	{attribute 'TcIecLibraryType'}
	{attribute 'external_name' := 'F_VN_MeasureAngleBetweenEdgesExp_GUID_AE732A2F_0C2A_0A0F_674F_B2AA43375E72'}
	(* Measure the angle between 2 edges. *)
	FUNCTION F_VN_MeasureAngleBetweenEdgesExp : HRESULT
	VAR_INPUT
		ipSrcImage	:	ITcVnImage;	(* Source image (1 channel) *)
		fAngle	:	REFERENCE TO REAL;	(* Returns the angle between the detected edges (radians or degrees, depending on bAngleInDegrees) *)
		aInnerPoint	:	REFERENCE TO TcVnPoint2_REAL;	(* Position inside the angle to measure, from which to start the edge search process (in the direction of aOuterPoint1 and aOuterPoint2) *)
		aOuterPoint1	:	REFERENCE TO TcVnPoint2_REAL;	(* Position where the search process for edge 1 ends *)
		aOuterPoint2	:	REFERENCE TO TcVnPoint2_REAL;	(* Position where the search process for edge 2 ends *)
		eEdgeDirection	:	ETcVnEdgeDirection;	(* Specification of the edge direction from aInnerPoint to aOuterPoint1 and aOuterPoint2 to search for *)
		fMinStrength	:	REAL;	(* Specification of the minimum strength (intensity difference) of the edge to search for *)
		nSearchLines	:	UDINT;	(* Width of the search window, i.e. the number of search lines (3, 5, 7, ...), centered around the line specified by aInnerPoint and aOuterPoint1, aOuterPoint2 *)
		fSearchLineDist	:	REAL;	(* Distance between the search lines in pixels (> 0) *)
		nMaxThickness	:	UDINT;	(* Specification of the maximum thickness of the edge to search for, which means fMinStrength must be reached within nMaxThickness pixels *)
		bInvertSearchDirection	:	BOOL;	(* If true, the search starts from each aOuterPoint in direction of aInnerPoint *)
		nSubpixelsIterations	:	UDINT;	(* Specifies the number of subpixels (for INTERPOLATION, 10 - 20 usually is sufficient) or maximum number of iterations for optimizing the parameters (for APPROX_ERF and APPROX_GAUSSIAN, 50 - 100 usually is sufficient) *)
		bAngleInDegrees	:	BOOL;	(* fAngle is in degrees, if true *)
		fApproxPrecision	:	REAL;	(* Specifies the approximation precision for APPROX_ERF and APPROX_GAUSSIAN (0.001 usually is sufficient, unused for INTERPOLATION) *)
		eAlgorithm	:	ETcVnEdgeDetectionAlgorithm;	(* Selection of the edge detection algorithm *)
		ipEdgePoints1	:	REFERENCE TO ITcVnContainer;	(* Returns the detected edge points between aInnerPoint and aOuterPoint1 (ContainerType_Vector_TcVnPoint2_REAL) *)
		ipEdgePoints2	:	REFERENCE TO ITcVnContainer;	(* Returns the detected edge points between aInnerPoint and aOuterPoint2 (ContainerType_Vector_TcVnPoint2_REAL) *)
		hrPrev	:	HRESULT;	(* HRESULT indicating the result of previous operations (If SUCCEEDED(hrPrev) equals false, no operation is executed.) *)
	END_VAR

END_FUNCTION

// Functions/Measurement/F_VN_MeasureEdgeDistance

	{attribute 'TcIecLibraryType'}
	{attribute 'external_name' := 'F_VN_MeasureEdgeDistance_GUID_7CBEE0F0_467B_0047_5A97_FA055498E2F6'}
	(* Measure the distance between 2 parallel edges, using an interpolation method. *)
	FUNCTION F_VN_MeasureEdgeDistance : HRESULT
	VAR_INPUT
		ipSrcImage	:	ITcVnImage;	(* Source image (1 channel) *)
		fAvgDistance	:	REFERENCE TO REAL;	(* Returns the average distance between the detected edges *)
		aStartPoint	:	REFERENCE TO TcVnPoint2_REAL;	(* Position from which to start the search process (in the direction of aEndPoint) *)
		aEndPoint	:	REFERENCE TO TcVnPoint2_REAL;	(* Position where the search process ends *)
		eEdgeDirection	:	ETcVnEdgeDirection;	(* Specification of the edge direction from aStartPoint to aEndPoint to search for *)
		fMinStrength	:	REAL;	(* Specification of the minimum strength (intensity difference) of the edge to search for *)
		nSearchLines	:	UDINT;	(* Width of the search window, i.e. the number of search lines (1, 3, 5, 7, ...), centered around the line specified by aStartPoint and aEndPoint *)
		hrPrev	:	HRESULT;	(* HRESULT indicating the result of previous operations (If SUCCEEDED(hrPrev) equals false, no operation is executed.) *)
	END_VAR

END_FUNCTION

// Functions/Measurement/F_VN_MeasureEdgeDistanceExp

	{attribute 'TcIecLibraryType'}
	{attribute 'external_name' := 'F_VN_MeasureEdgeDistanceExp_GUID_A22933CA_C8EC_0EED_56A6_BA58A31C374F'}
	(* Measure the distance between 2 parallel edges. (expert function) *)
	FUNCTION F_VN_MeasureEdgeDistanceExp : HRESULT
	VAR_INPUT
		ipSrcImage	:	ITcVnImage;	(* Source image (1 channel) *)
		fAvgDistance	:	REFERENCE TO REAL;	(* Returns the average distance between the detected edges *)
		aStartPoint	:	REFERENCE TO TcVnPoint2_REAL;	(* Position from which to start the search process (in the direction of aEndPoint) *)
		aEndPoint	:	REFERENCE TO TcVnPoint2_REAL;	(* Position where the search process ends *)
		eEdgeDirection	:	ETcVnEdgeDirection;	(* Specification of the edge direction from aStartPoint to aEndPoint to search for *)
		fMinStrength	:	REAL;	(* Specification of the minimum strength (intensity difference) of the edge to search for *)
		nSearchLines	:	UDINT;	(* Width of the search window, i.e. the number of search lines (1, 3, 5, 7, ...), centered around the line specified by aStartPoint and aEndPoint *)
		fSearchLineDist	:	REAL;	(* Distance between the search lines in pixels (> 0) *)
		nMaxThickness	:	UDINT;	(* Specification of the maximum thickness of the edge to search for, which means fMinStrength must be reached within nMaxThickness pixels *)
		bInvertSearchDirection	:	BOOL;	(* If true, the search starts from the center point between aStartPoint and aEndPoint in both directions *)
		fSearchGap	:	REAL;	(* Optional width of a gap (>= 0, centered between aStartPoint and aEndPoint), that is neglected for searching edges (can reduce execution time). The 2 edges to search for must be on different sides of the gap. *)
		nSubpixelsIterations	:	UDINT;	(* Specifies the number of subpixels (for INTERPOLATION, 10 - 20 usually is sufficient) or maximum number of iterations for optimizing the parameters (for APPROX_ERF and APPROX_GAUSSIAN, 50 - 100 usually is sufficient) *)
		fApproxPrecision	:	REAL;	(* Specifies the approximation precision for APPROX_ERF and APPROX_GAUSSIAN (0.001 usually is sufficient, unused for INTERPOLATION) *)
		eAlgorithm	:	ETcVnEdgeDetectionAlgorithm;	(* Selection of the edge detection algorithm *)
		ipEdgePoints1	:	REFERENCE TO ITcVnContainer;	(* Returns the detected edge points of the edge near aStartPoint (optional, set to 0 if not required; ContainerType_Vector_TcVnPoint2_REAL) *)
		ipEdgePoints2	:	REFERENCE TO ITcVnContainer;	(* Returns the detected edge points of the edge near aEndPoint (optional, set to 0 if not required; ContainerType_Vector_TcVnPoint2_REAL) *)
		ipDistances	:	REFERENCE TO ITcVnContainer;	(* Returns the distances between the detected edge points (optional, set to 0 if not required; ContainerType_Vector_REAL) *)
		hrPrev	:	HRESULT;	(* HRESULT indicating the result of previous operations (If SUCCEEDED(hrPrev) equals false, no operation is executed.) *)
	END_VAR

END_FUNCTION

// Functions/Measurement/F_VN_MeasureMinEdgeDistance

	{attribute 'TcIecLibraryType'}
	{attribute 'external_name' := 'F_VN_MeasureMinEdgeDistance_GUID_BAEABED5_95CB_0A35_52C1_670B9836C077'}
	(* Measure the minimum distance within the specified search window between 2 edges, using an interpolation method. *)
	FUNCTION F_VN_MeasureMinEdgeDistance : HRESULT
	VAR_INPUT
		ipSrcImage	:	ITcVnImage;	(* Source image (1 channel) *)
		fMinDistance	:	REFERENCE TO REAL;	(* Returns the minimum distance between the detected edges *)
		aStartPoint	:	REFERENCE TO TcVnPoint2_REAL;	(* Position from which to start the search process (in the direction of aEndPoint) *)
		aEndPoint	:	REFERENCE TO TcVnPoint2_REAL;	(* Position where the search process ends *)
		eEdgeDirection	:	ETcVnEdgeDirection;	(* Specification of the edge direction from aStartPoint to aEndPoint to search for *)
		fMinStrength	:	REAL;	(* Specification of the minimum strength (intensity difference) of the edge to search for *)
		nSearchLines	:	UDINT;	(* Width of the search window, i.e. the number of search lines (1, 3, 5, 7, ...), centered around the line specified by aStartPoint and aEndPoint *)
		hrPrev	:	HRESULT;	(* HRESULT indicating the result of previous operations (If SUCCEEDED(hrPrev) equals false, no operation is executed.) *)
	END_VAR

END_FUNCTION

// Functions/Measurement/F_VN_MeasureMinEdgeDistanceExp

	{attribute 'TcIecLibraryType'}
	{attribute 'external_name' := 'F_VN_MeasureMinEdgeDistanceExp_GUID_0C472EFC_B706_0DF3_5CDC_D468A697A380'}
	(* Measure the minimum distance within the specified search window between 2 edges. (expert function) *)
	FUNCTION F_VN_MeasureMinEdgeDistanceExp : HRESULT
	VAR_INPUT
		ipSrcImage	:	ITcVnImage;	(* Source image (1 channel) *)
		fMinDistance	:	REFERENCE TO REAL;	(* Returns the minimum distance between the detected edges *)
		aStartPoint	:	REFERENCE TO TcVnPoint2_REAL;	(* Position from which to start the search process (in the direction of aEndPoint) *)
		aEndPoint	:	REFERENCE TO TcVnPoint2_REAL;	(* Position where the search process ends *)
		eEdgeDirection	:	ETcVnEdgeDirection;	(* Specification of the edge direction from aStartPoint to aEndPoint to search for *)
		fMinStrength	:	REAL;	(* Specification of the minimum strength (intensity difference) of the edge to search for *)
		nSearchLines	:	UDINT;	(* Width of the search window, i.e. the number of search lines (1, 3, 5, 7, ...), centered around the line specified by aStartPoint and aEndPoint *)
		fSearchLineDist	:	REAL;	(* Distance between the search lines in pixels (> 0) *)
		nMaxThickness	:	UDINT;	(* Specification of the maximum thickness of the edge to search for, which means fMinStrength must be reached within nMaxThickness pixels *)
		bInvertSearchDirection	:	BOOL;	(* If true, the search starts from the center point between aStartPoint and aEndPoint in both directions *)
		fSearchGap	:	REAL;	(* Optional width of a gap (>= 0, centered between aStartPoint and aEndPoint), that is neglected for searching edges (can reduce execution time). The 2 edges to search for must be on different sides of the gap. *)
		nSubpixelsIterations	:	UDINT;	(* Specifies the number of subpixels (for INTERPOLATION, 10 - 20 usually is sufficient) or maximum number of iterations for optimizing the parameters (for APPROX_ERF and APPROX_GAUSSIAN, 50 - 100 usually is sufficient) *)
		fApproxPrecision	:	REAL;	(* Specifies the approximation precision for APPROX_ERF and APPROX_GAUSSIAN (0.001 usually is sufficient, unused for INTERPOLATION) *)
		eAlgorithm	:	ETcVnEdgeDetectionAlgorithm;	(* Selection of the edge detection algorithm *)
		ipEdgePoints1	:	REFERENCE TO ITcVnContainer;	(* Returns the detected edge points of the edge near aStartPoint (optional, set to 0 if not required; ContainerType_Vector_TcVnPoint2_REAL) *)
		ipEdgePoints2	:	REFERENCE TO ITcVnContainer;	(* Returns the detected edge points of the edge near aEndPoint (optional, set to 0 if not required; ContainerType_Vector_TcVnPoint2_REAL) *)
		aPoint1	:	REFERENCE TO TcVnPoint2_REAL;	(* Returns the point on the edge near aStartPoint, for which the minimum distance is achieved *)
		aPoint2	:	REFERENCE TO TcVnPoint2_REAL;	(* Returns the point on the edge near aEndPoint, for which the minimum distance is achieved *)
		hrPrev	:	HRESULT;	(* HRESULT indicating the result of previous operations (If SUCCEEDED(hrPrev) equals false, no operation is executed.) *)
	END_VAR

END_FUNCTION

// Functions/Basic Container Operations/F_VN_AdvanceIterator

	{attribute 'TcIecLibraryType'}
	{attribute 'external_name' := 'F_VN_AdvanceIterator_GUID_ACC8E97D_98FD_0CAF_65B6_42FD1B5BC612'}
	(* Advance an iterator by the specified offset. *)
	FUNCTION F_VN_AdvanceIterator : HRESULT
	VAR_INPUT
		ipIterator	:	ITcVnForwardIterator;	(* Iterator to be advanced *)
		nOffset	:	LINT;	(* Offset, by which ipIterator is advanced *)
		hrPrev	:	HRESULT;	(* HRESULT indicating the result of previous operations (If SUCCEEDED(hrPrev) equals false, no operation is executed.) *)
	END_VAR

END_FUNCTION

// Functions/Basic Container Operations/F_VN_CheckIfEmpty

	{attribute 'TcIecLibraryType'}
	{attribute 'external_name' := 'F_VN_CheckIfEmpty_GUID_F72A904D_F5AF_0726_5092_69B65BB6D2D0'}
	(* Checks if the container is empty. (Alternatively use interface method .CheckIfEmpty.) *)
	FUNCTION F_VN_CheckIfEmpty : HRESULT
	VAR_INPUT
		ipContainer	:	ITcVnContainer;	(* Container *)
		hrPrev	:	HRESULT;	(* HRESULT indicating the result of previous operations (If SUCCEEDED(hrPrev) equals false, no operation is executed.) *)
	END_VAR

END_FUNCTION

// Functions/Basic Container Operations/F_VN_CheckIfIteratorIsAtEnd

	{attribute 'TcIecLibraryType'}
	{attribute 'external_name' := 'F_VN_CheckIfIteratorIsAtEnd_GUID_30C2C0F0_70D6_0795_4B1A_E8C5B6524E93'}
	(* Checks if the iterator points to the past-the-end element. (Alternatively use interface method .CheckIfEnd.) *)
	FUNCTION F_VN_CheckIfIteratorIsAtEnd : HRESULT
	VAR_INPUT
		ipIterator	:	ITcVnForwardIterator;	(* Iterator *)
		hrPrev	:	HRESULT;	(* HRESULT indicating the result of previous operations (If SUCCEEDED(hrPrev) equals false, no operation is executed.) *)
	END_VAR

END_FUNCTION

// Functions/Basic Container Operations/F_VN_ConvertContainerType

	{attribute 'TcIecLibraryType'}
	{attribute 'external_name' := 'F_VN_ConvertContainerType_GUID_01A1FD6A_9814_007F_619D_D5C12B443F08'}
	(* Converts a container to another type (Struct element types are not supported). *)
	FUNCTION F_VN_ConvertContainerType : HRESULT
	VAR_INPUT
		ipSrcContainer	:	ITcVnContainer;	(* Source container *)
		ipDestContainer	:	REFERENCE TO ITcVnContainer;	(* Returns the converted container *)
		nDestTypeGuid	:	GUID;	(* Specifies the destination container type for the conversion *)
		hrPrev	:	HRESULT;	(* HRESULT indicating the result of previous operations (If SUCCEEDED(hrPrev) equals false, no operation is executed.) *)
	END_VAR

END_FUNCTION

// Functions/Basic Container Operations/F_VN_CopyContainer

	{attribute 'TcIecLibraryType'}
	{attribute 'external_name' := 'F_VN_CopyContainer_GUID_DAA3A3C5_5EBA_03BD_7F09_6558B2F826E3'}
	(* Copys a container. *)
	FUNCTION F_VN_CopyContainer : HRESULT
	VAR_INPUT
		ipSrcContainer	:	ITcVnContainer;	(* Source container *)
		ipDestContainer	:	REFERENCE TO ITcVnContainer;	(* Destination container (same type ID as ipSrcContainer; Non-zero interface pointers are reused.) *)
		hrPrev	:	HRESULT;	(* HRESULT indicating the result of previous operations (If SUCCEEDED(hrPrev) equals false, no operation is executed.) *)
	END_VAR

END_FUNCTION

// Functions/Basic Container Operations/F_VN_CopyContainerElementsConditional_ITcVnContainer

	{attribute 'TcIecLibraryType'}
	{attribute 'external_name' := 'F_VN_CopyContainerElementsConditional_ITcVnContainer_GUID_2F464D18_7218_035A_4EBD_E5C0F488799D'}
	(* Copys container elements to a new container, depending on a custom condition. *)
	FUNCTION F_VN_CopyContainerElementsConditional_ITcVnContainer : HRESULT
	VAR_INPUT
		ipSrcContainer	:	ITcVnContainer;	(* Source container *)
		ipDestContainer	:	REFERENCE TO ITcVnContainer;	(* Returns a container with elements, that match the condition *)
		ipConditionFB	:	ITcVnCustomElementCondition_ITcVnContainer;	(* Custom condition *)
		hrPrev	:	HRESULT;	(* HRESULT indicating the result of previous operations (If SUCCEEDED(hrPrev) equals false, no operation is executed.) *)
	END_VAR

END_FUNCTION

// Interfaces/Containers/Function Blocks/ITcVnCustomElementCondition_ITcVnContainer

	(* Offers an interface for a custom condition computed for a container. *)
	{attribute 'c++_compatible'}
	INTERFACE ITcVnCustomElementCondition_ITcVnContainer


(* Evaluates the condition for the container. *)
	{attribute 'c++_compatible'}
	{attribute 'minimal_input_size' := '4'}
	{attribute 'pack_mode' := '4'}
	METHOD Condition : BOOL
	VAR_INPUT
		ipElement : ITcVnContainer;
	END_VAR
END_METHOD

END_INTERFACE

// Functions/Basic Container Operations/F_VN_CopyContainerElementsConditional_ITcVnForwardIterator

	{attribute 'TcIecLibraryType'}
	{attribute 'external_name' := 'F_VN_CopyContainerElementsConditional_ITcVnForwardIterator_GUID_435C1609_A638_0537_49B4_06CAF8EA0EB5'}
	(* Copys container elements to a new container, depending on a custom condition. *)
	FUNCTION F_VN_CopyContainerElementsConditional_ITcVnForwardIterator : HRESULT
	VAR_INPUT
		ipSrcContainer	:	ITcVnContainer;	(* Source container *)
		ipDestContainer	:	REFERENCE TO ITcVnContainer;	(* Returns a container with elements, that match the condition *)
		ipConditionFB	:	ITcVnCustomElementCondition_ITcVnForwardIterator;	(* Custom condition *)
		hrPrev	:	HRESULT;	(* HRESULT indicating the result of previous operations (If SUCCEEDED(hrPrev) equals false, no operation is executed.) *)
	END_VAR

END_FUNCTION

// Interfaces/Containers/Function Blocks/ITcVnCustomElementCondition_ITcVnForwardIterator

	(* Offers an interface for a custom condition computed for an element represented by an ITcVnForwardIterator. *)
	{attribute 'c++_compatible'}
	INTERFACE ITcVnCustomElementCondition_ITcVnForwardIterator


(* Evaluates the condition for the provided element. *)
	{attribute 'c++_compatible'}
	{attribute 'minimal_input_size' := '4'}
	{attribute 'pack_mode' := '4'}
	METHOD Condition : BOOL
	VAR_INPUT
		ipElement : ITcVnForwardIterator;
	END_VAR
END_METHOD

END_INTERFACE

// Functions/Basic Container Operations/F_VN_CreateContainer

	{attribute 'TcIecLibraryType'}
	{attribute 'external_name' := 'F_VN_CreateContainer_GUID_61D37913_CA0D_07D0_5304_6E5DDCD021C0'}
	(* Creates a container with type GUID nTypeGuid and return its container interface. *)
	FUNCTION F_VN_CreateContainer : HRESULT
	VAR_INPUT
		ipContainer	:	REFERENCE TO ITcVnContainer;	(* Returns the created container *)
		nTypeGuid	:	GUID;	(* Type GUID of the container to be created *)
		nElementNum	:	ULINT;	(* Number of elements *)
		hrPrev	:	HRESULT;	(* HRESULT indicating the result of previous operations (If SUCCEEDED(hrPrev) equals false, no operation is executed.) *)
	END_VAR

END_FUNCTION

// Functions/Basic Container Operations/F_VN_CreateContainerFromArray

	{attribute 'TcIecLibraryType'}
	{attribute 'external_name' := 'F_VN_CreateContainerFromArray_GUID_AA5B3DDF_00B1_0B21_7AD4_970908632B01'}
	(* Creates a container with type GUID nTypeGuid, initialize it with provided data and return its container interface. Only supported for basic container types, i.e. not for containers of containers. *)
	FUNCTION F_VN_CreateContainerFromArray : HRESULT
	VAR_INPUT
		pData	:	PVOID;	(* Pointer to the data array. Make sure that the array contains at least nElementNum elements and that the array element type matches the container element type. *)
		ipContainer	:	REFERENCE TO ITcVnContainer;	(* Returns the created container *)
		nTypeGuid	:	GUID;	(* Type GUID of the container to be created *)
		nElementNum	:	ULINT;	(* Number of elements to copy from pData *)
		hrPrev	:	HRESULT;	(* HRESULT indicating the result of previous operations (If SUCCEEDED(hrPrev) equals false, no operation is executed.) *)
	END_VAR

END_FUNCTION

// Functions/Basic Container Operations/F_VN_EraseFromContainer

	{attribute 'TcIecLibraryType'}
	{attribute 'external_name' := 'F_VN_EraseFromContainer_GUID_D686421B_0E77_0897_58AA_85FC33B178E9'}
	(* Erase elements from a container. *)
	FUNCTION F_VN_EraseFromContainer : HRESULT
	VAR_INPUT
		ipContainer	:	ITcVnContainer;	(* Container from which to erase elements *)
		nStartIdx	:	ULINT;	(* Index of the first element to erase *)
		nCount	:	ULINT;	(* Number of elements to erase *)
		hrPrev	:	HRESULT;	(* HRESULT indicating the result of previous operations (If SUCCEEDED(hrPrev) equals false, no operation is executed.) *)
	END_VAR

END_FUNCTION

// Functions/Basic Container Operations/F_VN_ExportContainer

	{attribute 'TcIecLibraryType'}
	{attribute 'external_name' := 'F_VN_ExportContainer_GUID_B3105DE8_989A_095E_6EB1_2DCFC3551E31'}
	(* Export the container elements into a buffer (e.g. an array). Only possible for containers with basic elements. *)
	FUNCTION F_VN_ExportContainer : HRESULT
	VAR_INPUT
		ipContainer	:	ITcVnContainer;	(* Container with basic elements *)
		pBuffer	:	PVOID;	(* Buffer to store the container elements (Make sure to allocate enough memory! The required size in bytes can be determined using the function F_VN_ExportContainerSize) *)
		nBufferSize	:	ULINT;	(* Size of the buffer memory in bytes *)
		hrPrev	:	HRESULT;	(* HRESULT indicating the result of previous operations (If SUCCEEDED(hrPrev) equals false, no operation is executed.) *)
	END_VAR

END_FUNCTION

// Functions/Basic Container Operations/F_VN_ExportContainerSize

	{attribute 'TcIecLibraryType'}
	{attribute 'external_name' := 'F_VN_ExportContainerSize_GUID_76F4BBB5_BAC4_061D_63B1_EE647B621371'}
	(* Determine the required buffer size in bytes to store all container elements (number_of_Elements * size_per_Element). Only possible for containers with basic elements. *)
	FUNCTION F_VN_ExportContainerSize : HRESULT
	VAR_INPUT
		ipContainer	:	ITcVnContainer;	(* Container with basic elements *)
		nBufferSize	:	REFERENCE TO ULINT;	(* Output parameter containing the required buffer size *)
		hrPrev	:	HRESULT;	(* HRESULT indicating the result of previous operations (If SUCCEEDED(hrPrev) equals false, no operation is executed.) *)
	END_VAR

END_FUNCTION

// Functions/Basic Container Operations/F_VN_ExportContainer_String

	{attribute 'TcIecLibraryType'}
	{attribute 'external_name' := 'F_VN_ExportContainer_String_GUID_5BD8ABC1_1BA1_0734_5AF1_0620F612769A'}
	(* Export the container elements into a string. Only possible for containers of type ContainerType_String_SINT. *)
	FUNCTION F_VN_ExportContainer_String : HRESULT
	VAR_INPUT
		ipContainer	:	ITcVnContainer;	(* Container of type ContainerType_String_SINT *)
	END_VAR
	VAR_IN_OUT CONSTANT
		sText	:	STRING;	(* Make sure to choose a sufficient STRING size! The required size can be determined using the function VnExportContainerSize. *)
	END_VAR
	VAR_INPUT
		nMaxLength	:	ULINT;	(* Maximum string length to export (including 0 termination). If the container content is longer, the string is cut off at nMaxLength - 1 and 0 termination is appended. In this case, S_FALSE is returned. *)
		hrPrev	:	HRESULT;	(* HRESULT indicating the result of previous operations (If SUCCEEDED(hrPrev) equals false, no operation is executed.) *)
	END_VAR

END_FUNCTION

// Functions/Basic Container Operations/F_VN_ExportSubContainer

	{attribute 'TcIecLibraryType'}
	{attribute 'external_name' := 'F_VN_ExportSubContainer_GUID_2C76D183_CD1A_0BBB_4C3C_54CD9386FE08'}
	(* Export the container elements of a sub-container into a buffer (e.g. an array). Only possible for 2-dimensional containers with basic elements. *)
	FUNCTION F_VN_ExportSubContainer : HRESULT
	VAR_INPUT
		ipContainer	:	ITcVnContainer;	(* Container with basic elements *)
		nIndex	:	ULINT;	(* Index of the requested element *)
		pBuffer	:	PVOID;	(* Buffer to store the container elements (Make sure to allocate enough memory! The required size in bytes can be determined using the function F_VN_ExportSubContainerSize) *)
		nBufferSize	:	ULINT;	(* Size of the buffer memory in bytes *)
		hrPrev	:	HRESULT;	(* HRESULT indicating the result of previous operations (If SUCCEEDED(hrPrev) equals false, no operation is executed.) *)
	END_VAR

END_FUNCTION

// Functions/Basic Container Operations/F_VN_ExportSubContainerSize

	{attribute 'TcIecLibraryType'}
	{attribute 'external_name' := 'F_VN_ExportSubContainerSize_GUID_9A378173_3E8F_041B_7D7A_DBB1303321B8'}
	(* Determine the required buffer size in bytes to store all container elements of a sub-container (number_of_Elements * size_per_Element). Only possible for 2-dimensional containers with basic elements. *)
	FUNCTION F_VN_ExportSubContainerSize : HRESULT
	VAR_INPUT
		ipContainer	:	ITcVnContainer;	(* Container with basic elements *)
		nIndex	:	ULINT;	(* Index of the requested element *)
		nBufferSize	:	REFERENCE TO ULINT;	(* Output parameter containing the required buffer size *)
		hrPrev	:	HRESULT;	(* HRESULT indicating the result of previous operations (If SUCCEEDED(hrPrev) equals false, no operation is executed.) *)
	END_VAR

END_FUNCTION

// Functions/Basic Container Operations/F_VN_ExportSubContainer_String

	{attribute 'TcIecLibraryType'}
	{attribute 'external_name' := 'F_VN_ExportSubContainer_String_GUID_4F555A08_F7D7_0928_7E2C_5AC3BF1C3727'}
	(* Export the container elements of a sub-container into a string. Only possible for 2-dimensional containers of type ContainerType_Vector_String_SINT. *)
	FUNCTION F_VN_ExportSubContainer_String : HRESULT
	VAR_INPUT
		ipContainer	:	ITcVnContainer;	(* Container of type ContainerType_Vector_String_SINT *)
		nIndex	:	ULINT;	(* Index of the requested element *)
	END_VAR
	VAR_IN_OUT CONSTANT
		sText	:	STRING;	(* Make sure to choose a sufficient STRING size! The required size can be determined using the function VnExportSubContainerSize. *)
	END_VAR
	VAR_INPUT
		nMaxLength	:	ULINT;	(* Maximum string length to export (including 0 termination). If the container content is longer, the string is cut off at nMaxLength - 1 and 0 termination is appended. In this case, S_FALSE is returned. *)
		hrPrev	:	HRESULT;	(* HRESULT indicating the result of previous operations (If SUCCEEDED(hrPrev) equals false, no operation is executed.) *)
	END_VAR

END_FUNCTION

// Functions/Basic Container Operations/F_VN_ExtractContainerRange

	{attribute 'TcIecLibraryType'}
	{attribute 'external_name' := 'F_VN_ExtractContainerRange_GUID_4EB284E8_0B53_0D83_5DCE_29B545B8D0A0'}
	(* Copy the specified range of the source container into the destination container. (If the destination container already contains elements, they will be removed.) *)
	FUNCTION F_VN_ExtractContainerRange : HRESULT
	VAR_INPUT
		ipSrcContainer	:	ITcVnContainer;	(* Source container *)
		ipDestContainer	:	REFERENCE TO ITcVnContainer;	(* Destination container *)
		nFirstIdx	:	ULINT;	(* Index of the first element to copy *)
		nLastIdx	:	ULINT;	(* Index of the last element to copy *)
		hrPrev	:	HRESULT;	(* HRESULT indicating the result of previous operations (If SUCCEEDED(hrPrev) equals false, no operation is executed.) *)
	END_VAR

END_FUNCTION

// Functions/Basic Container Operations/F_VN_GetContainer

	{attribute 'TcIecLibraryType'}
	{attribute 'external_name' := 'F_VN_GetContainer_GUID_27505B6E_9EAE_086D_5BCA_CC9172BAFD0B'}
	(* Gets a pointer to the current element converted into an ITcVnContainer interface and increment its reference counter (only possible for container types). (Alternatively use interface method .GetContainer.) *)
	FUNCTION F_VN_GetContainer : HRESULT
	VAR_INPUT
		ipIterator	:	ITcVnForwardIterator;	(* Iterator *)
		ipContainer	:	REFERENCE TO ITcVnContainer;	(* Returns the container interface *)
		hrPrev	:	HRESULT;	(* HRESULT indicating the result of previous operations (If SUCCEEDED(hrPrev) equals false, no operation is executed.) *)
	END_VAR

END_FUNCTION

// Functions/Basic Container Operations/F_VN_GetContainerExp

	{attribute 'TcIecLibraryType'}
	{attribute 'external_name' := 'F_VN_GetContainerExp_GUID_436CF1E3_F353_08D3_710A_C75CD81D8DEB'}
	(* Gets a pointer to the current element converted into an ITcVnContainer interface and increment its reference counter (only possible for container types). Additionally, an offset to increment or decrement the iterator afterwards can be provided. (expert function) *)
	FUNCTION F_VN_GetContainerExp : HRESULT
	VAR_INPUT
		ipIterator	:	ITcVnForwardIterator;	(* Iterator *)
		ipContainer	:	REFERENCE TO ITcVnContainer;	(* Returns the container interface *)
		nOffset	:	DINT;	(* Offset to increment (>0) or decrement (<0) the iterator afterwards *)
		hrPrev	:	HRESULT;	(* HRESULT indicating the result of previous operations (If SUCCEEDED(hrPrev) equals false, no operation is executed.) *)
	END_VAR

END_FUNCTION

// Functions/Basic Container Operations/F_VN_GetForwardIterator

	{attribute 'TcIecLibraryType'}
	{attribute 'external_name' := 'F_VN_GetForwardIterator_GUID_43078F70_57B1_0E73_4856_F4D286EF9EA2'}
	(* Gets a forward iterator for the container. (Alternatively use interface method .GetForwardIterator.) *)
	FUNCTION F_VN_GetForwardIterator : HRESULT
	VAR_INPUT
		ipContainer	:	ITcVnContainer;	(* Container *)
		ipIterator	:	REFERENCE TO ITcVnForwardIterator;	(* Returns the iterator interface *)
		hrPrev	:	HRESULT;	(* HRESULT indicating the result of previous operations (If SUCCEEDED(hrPrev) equals false, no operation is executed.) *)
	END_VAR

END_FUNCTION

// Functions/Basic Container Operations/F_VN_GetNumberOfElements

	{attribute 'TcIecLibraryType'}
	{attribute 'external_name' := 'F_VN_GetNumberOfElements_GUID_C1684A08_CB59_09CF_7B51_7659520AA3E9'}
	(* Gets the number of elements in the container. (Alternatively use interface method .getElementNum.) *)
	FUNCTION F_VN_GetNumberOfElements : HRESULT
	VAR_INPUT
		ipContainer	:	ITcVnContainer;	(* Container *)
		nNumberOfElements	:	REFERENCE TO ULINT;	(* Returns the number of elements in ipContainer *)
		hrPrev	:	HRESULT;	(* HRESULT indicating the result of previous operations (If SUCCEEDED(hrPrev) equals false, no operation is executed.) *)
	END_VAR

END_FUNCTION

// Functions/Basic Container Operations/F_VN_GetRandomAccessIterator

	{attribute 'TcIecLibraryType'}
	{attribute 'external_name' := 'F_VN_GetRandomAccessIterator_GUID_3FA92340_67E8_032A_7ED0_6A69355C56A7'}
	(* Gets a random access iterator for the container. (Alternatively use interface method .GetRandomAccessIterator.) *)
	FUNCTION F_VN_GetRandomAccessIterator : HRESULT
	VAR_INPUT
		ipContainer	:	ITcVnContainer;	(* Container *)
		ipIterator	:	REFERENCE TO ITcVnRandomAccessIterator;	(* Returns the iterator interface *)
		hrPrev	:	HRESULT;	(* HRESULT indicating the result of previous operations (If SUCCEEDED(hrPrev) equals false, no operation is executed.) *)
	END_VAR

END_FUNCTION

// Functions/Basic Container Operations/F_VN_IncrementIterator

	{attribute 'TcIecLibraryType'}
	{attribute 'external_name' := 'F_VN_IncrementIterator_GUID_69A16AA6_5F55_058E_6ED7_D592BD9145A4'}
	(* Increment the iterator. (Alternatively use interface method .Increment.) *)
	FUNCTION F_VN_IncrementIterator : HRESULT
	VAR_INPUT
		ipIterator	:	ITcVnForwardIterator;	(* Iterator *)
		hrPrev	:	HRESULT;	(* HRESULT indicating the result of previous operations (If SUCCEEDED(hrPrev) equals false, no operation is executed.) *)
	END_VAR

END_FUNCTION

// Functions/Basic Container Operations/F_VN_IteratorDistance

	{attribute 'TcIecLibraryType'}
	{attribute 'external_name' := 'F_VN_IteratorDistance_GUID_DC10392B_7965_07D5_51DE_916FCBD58C32'}
	(* Computes the distance between 2 iterators. *)
	FUNCTION F_VN_IteratorDistance : HRESULT
	VAR_INPUT
		ipIteratorFirst	:	ITcVnForwardIterator;	(* First iterator *)
		ipIteratorLast	:	ITcVnForwardIterator;	(* Last iterator *)
		nDistance	:	REFERENCE TO LINT;	(* Returns the computed distance *)
		hrPrev	:	HRESULT;	(* HRESULT indicating the result of previous operations (If SUCCEEDED(hrPrev) equals false, no operation is executed.) *)
	END_VAR

END_FUNCTION

// Functions/Basic Container Operations/F_VN_ReserveContainerMemory

	{attribute 'TcIecLibraryType'}
	{attribute 'external_name' := 'F_VN_ReserveContainerMemory_GUID_A6C96216_5A91_0611_6333_23BBD3722D9C'}
	(* Reserve container memory (call with maximum required number of elements before manually appending elements for better performance) *)
	FUNCTION F_VN_ReserveContainerMemory : HRESULT
	VAR_INPUT
		ipContainer	:	ITcVnContainer;	(* Container for which to reserve the memory *)
		nElements	:	ULINT;	(* Number of elements for which the container should reserve memory *)
		hrPrev	:	HRESULT;	(* HRESULT indicating the result of previous operations (If SUCCEEDED(hrPrev) equals false, no operation is executed.) *)
	END_VAR

END_FUNCTION

// Functions/Basic Container Operations/F_VN_ReverseContainer

	{attribute 'TcIecLibraryType'}
	{attribute 'external_name' := 'F_VN_ReverseContainer_GUID_35F112E5_387D_0B85_557A_AEA6C3B2DB12'}
	(* Reverse the container elements. *)
	FUNCTION F_VN_ReverseContainer : HRESULT
	VAR_INPUT
		ipContainer	:	ITcVnContainer;	(* Container to be reversed *)
		hrPrev	:	HRESULT;	(* HRESULT indicating the result of previous operations (If SUCCEEDED(hrPrev) equals false, no operation is executed.) *)
	END_VAR

END_FUNCTION

// Functions/Basic Container Operations/F_VN_SetContainer

	{attribute 'TcIecLibraryType'}
	{attribute 'external_name' := 'F_VN_SetContainer_GUID_E3937A25_D58C_09AB_7741_9A0CBC6B0412'}
	(* Sets the current element using an ITcVnContainer interface (only possible for container types). (Alternatively use interface method .SetContainer.) *)
	FUNCTION F_VN_SetContainer : HRESULT
	VAR_INPUT
		ipIterator	:	ITcVnForwardIterator;	(* Iterator *)
		ipContainer	:	ITcVnContainer;	(* Container interface of which the content is to be assigned to the current element *)
		hrPrev	:	HRESULT;	(* HRESULT indicating the result of previous operations (If SUCCEEDED(hrPrev) equals false, no operation is executed.) *)
	END_VAR

END_FUNCTION

// Functions/Basic Container Operations/F_VN_SetIteratorToBegin

	{attribute 'TcIecLibraryType'}
	{attribute 'external_name' := 'F_VN_SetIteratorToBegin_GUID_51E4D889_EE17_05C3_44C3_7A5207251AFA'}
	(* Sets the iterator to the first element of the container. (Alternatively use interface method .SetToBegin.) *)
	FUNCTION F_VN_SetIteratorToBegin : HRESULT
	VAR_INPUT
		ipIterator	:	ITcVnForwardIterator;	(* Iterator *)
		hrPrev	:	HRESULT;	(* HRESULT indicating the result of previous operations (If SUCCEEDED(hrPrev) equals false, no operation is executed.) *)
	END_VAR

END_FUNCTION

// Functions/Geometric and Coordinate Transformations/F_VN_AlignRotatedImageRegion

	{attribute 'TcIecLibraryType'}
	{attribute 'external_name' := 'F_VN_AlignRotatedImageRegion_GUID_3F265FEA_BECE_014F_47AF_B5F8C6E76B10'}
	(* Copies the provided image region and aligns it to the image axes. *)
	FUNCTION F_VN_AlignRotatedImageRegion : HRESULT
	VAR_INPUT
		ipSrcImage	:	ITcVnImage;	(* Source image *)
		ipDestImage	:	REFERENCE TO ITcVnImage;	(* Destination image (An appropriate image will be created if required.) *)
		stRegion	:	REFERENCE TO TcVnRotatedRectangle;	(* Image region to be aligned *)
		hrPrev	:	HRESULT;	(* HRESULT indicating the result of previous operations (If SUCCEEDED(hrPrev) equals false, no operation is executed.) *)
	END_VAR

END_FUNCTION

// Functions/Geometric and Coordinate Transformations/F_VN_AlignRotatedImageRegionExp

	{attribute 'TcIecLibraryType'}
	{attribute 'external_name' := 'F_VN_AlignRotatedImageRegionExp_GUID_D33A5843_210C_0064_6EBC_CB88CD706C00'}
	(* Copies the provided image region and aligns it to the image axes. (expert function) *)
	FUNCTION F_VN_AlignRotatedImageRegionExp : HRESULT
	VAR_INPUT
		ipSrcImage	:	ITcVnImage;	(* Source image *)
		ipDestImage	:	REFERENCE TO ITcVnImage;	(* Destination image (An appropriate image will be created if required.) *)
		stRegion	:	REFERENCE TO TcVnRotatedRectangle;	(* Image region to be aligned *)
		eInterpolationType	:	ETcVnInterpolationType;	(* Interpolation method *)
		eBorderInterpolation	:	ETcVnBorderInterpolationMethod;	(* Border interpolation method (ISOLATED not supported) *)
		aBorderValue	:	REFERENCE TO TcVnVector4_LREAL;	(* Border value, if CONSTANT is used *)
		hrPrev	:	HRESULT;	(* HRESULT indicating the result of previous operations (If SUCCEEDED(hrPrev) equals false, no operation is executed.) *)
	END_VAR

END_FUNCTION

// Functions/Geometric and Coordinate Transformations/F_VN_ApplyRotationToAffineTransformation

	{attribute 'TcIecLibraryType'}
	{attribute 'external_name' := 'F_VN_ApplyRotationToAffineTransformation_GUID_D2AAEA5C_C5D3_0D46_678A_5DCA00EA5833'}
	(* Apply a rotation to an existing 2D affine transformation matrix. *)
	FUNCTION F_VN_ApplyRotationToAffineTransformation : HRESULT
	VAR_INPUT
		aTransformationMatrix	:	REFERENCE TO TcVnMatrix2x3_LREAL;	(* Affine transformation matrix to which the rotation is applied *)
		fAngle	:	LREAL;	(* Angle in radians (positive means counter-clockwise) *)
		hrPrev	:	HRESULT;	(* HRESULT indicating the result of previous operations (If SUCCEEDED(hrPrev) equals false, no operation is executed.) *)
	END_VAR

END_FUNCTION

// Functions/Geometric and Coordinate Transformations/F_VN_ApplyRotationToAffineTransformationExp

	{attribute 'TcIecLibraryType'}
	{attribute 'external_name' := 'F_VN_ApplyRotationToAffineTransformationExp_GUID_09811113_83D1_0FA5_740A_AEC9964AC26B'}
	(* Apply a rotation to an existing 2D affine transformation matrix. (expert function) *)
	FUNCTION F_VN_ApplyRotationToAffineTransformationExp : HRESULT
	VAR_INPUT
		aTransformationMatrix	:	REFERENCE TO TcVnMatrix2x3_LREAL;	(* Affine transformation matrix to which the rotation is applied *)
		fAngle	:	LREAL;	(* Angle in radians (positive means counter-clockwise) *)
		bUsePreMultiplication	:	BOOL;	(* Select if pre- or post-multiplication should be used *)
		hrPrev	:	HRESULT;	(* HRESULT indicating the result of previous operations (If SUCCEEDED(hrPrev) equals false, no operation is executed.) *)
	END_VAR

END_FUNCTION

// Functions/Geometric and Coordinate Transformations/F_VN_ApplyScalingToAffineTransformation

	{attribute 'TcIecLibraryType'}
	{attribute 'external_name' := 'F_VN_ApplyScalingToAffineTransformation_GUID_0AC37701_099D_0829_772F_D6736195BB34'}
	(* Apply a scaling to an existing 2D affine transformation matrix. *)
	FUNCTION F_VN_ApplyScalingToAffineTransformation : HRESULT
	VAR_INPUT
		aTransformationMatrix	:	REFERENCE TO TcVnMatrix2x3_LREAL;	(* Affine transformation matrix to which the scaling is applied *)
		fScaleX	:	LREAL;	(* Scaling factor in x direction *)
		fScaleY	:	LREAL;	(* Scaling factor in y direction *)
		hrPrev	:	HRESULT;	(* HRESULT indicating the result of previous operations (If SUCCEEDED(hrPrev) equals false, no operation is executed.) *)
	END_VAR

END_FUNCTION

// Functions/Geometric and Coordinate Transformations/F_VN_ApplyScalingToAffineTransformationExp

	{attribute 'TcIecLibraryType'}
	{attribute 'external_name' := 'F_VN_ApplyScalingToAffineTransformationExp_GUID_0B1DCD8E_602D_0379_4AFD_8BE184FF709D'}
	(* Apply a scaling to an existing 2D affine transformation matrix. (expert function) *)
	FUNCTION F_VN_ApplyScalingToAffineTransformationExp : HRESULT
	VAR_INPUT
		aTransformationMatrix	:	REFERENCE TO TcVnMatrix2x3_LREAL;	(* Affine transformation matrix to which the scaling is applied *)
		fScaleX	:	LREAL;	(* Scaling factor in x direction *)
		fScaleY	:	LREAL;	(* Scaling factor in y direction *)
		bUsePreMultiplication	:	BOOL;	(* Select if pre- or post-multiplication should be used *)
		hrPrev	:	HRESULT;	(* HRESULT indicating the result of previous operations (If SUCCEEDED(hrPrev) equals false, no operation is executed.) *)
	END_VAR

END_FUNCTION

// Functions/Geometric and Coordinate Transformations/F_VN_ApplyTranslationToAffineTransformation

	{attribute 'TcIecLibraryType'}
	{attribute 'external_name' := 'F_VN_ApplyTranslationToAffineTransformation_GUID_2CE336D6_8FF6_0659_73D0_7BE4ABCDC41C'}
	(* Apply a translation to an existing 2D affine transformation matrix. *)
	FUNCTION F_VN_ApplyTranslationToAffineTransformation : HRESULT
	VAR_INPUT
		aTransformationMatrix	:	REFERENCE TO TcVnMatrix2x3_LREAL;	(* Affine transformation matrix to which the translation is applied *)
		fDeltaX	:	LREAL;	(* Translation in x direction *)
		fDeltaY	:	LREAL;	(* Translation in y direction *)
		hrPrev	:	HRESULT;	(* HRESULT indicating the result of previous operations (If SUCCEEDED(hrPrev) equals false, no operation is executed.) *)
	END_VAR

END_FUNCTION

// Functions/Geometric and Coordinate Transformations/F_VN_ApplyTranslationToAffineTransformationExp

	{attribute 'TcIecLibraryType'}
	{attribute 'external_name' := 'F_VN_ApplyTranslationToAffineTransformationExp_GUID_B48E036C_FF70_0D75_7B83_23F5D06CED29'}
	(* Apply a translation to an existing 2D affine transformation matrix. (expert function) *)
	FUNCTION F_VN_ApplyTranslationToAffineTransformationExp : HRESULT
	VAR_INPUT
		aTransformationMatrix	:	REFERENCE TO TcVnMatrix2x3_LREAL;	(* Affine transformation matrix to which the translation is applied *)
		fDeltaX	:	LREAL;	(* Translation in x direction *)
		fDeltaY	:	LREAL;	(* Translation in y direction *)
		bUsePreMultiplication	:	BOOL;	(* Select if pre- or post-multiplication should be used *)
		hrPrev	:	HRESULT;	(* HRESULT indicating the result of previous operations (If SUCCEEDED(hrPrev) equals false, no operation is executed.) *)
	END_VAR

END_FUNCTION

// Functions/Geometric and Coordinate Transformations/F_VN_ApplyYAxisInversionToAffineTransformation

	{attribute 'TcIecLibraryType'}
	{attribute 'external_name' := 'F_VN_ApplyYAxisInversionToAffineTransformation_GUID_ABA7B922_0E85_0EC7_45FC_DB03AB370BB3'}
	(* Apply an inversion of the y-axis direction to an existing 2D affine transformation matrix. *)
	FUNCTION F_VN_ApplyYAxisInversionToAffineTransformation : HRESULT
	VAR_INPUT
		aTransformationMatrix	:	REFERENCE TO TcVnMatrix2x3_LREAL;	(* Affine transformation matrix to which the inversion of the y-axis direction is applied *)
		hrPrev	:	HRESULT;	(* HRESULT indicating the result of previous operations (If SUCCEEDED(hrPrev) equals false, no operation is executed.) *)
	END_VAR

END_FUNCTION

// Functions/Geometric and Coordinate Transformations/F_VN_ApplyYAxisInversionToAffineTransformationExp

	{attribute 'TcIecLibraryType'}
	{attribute 'external_name' := 'F_VN_ApplyYAxisInversionToAffineTransformationExp_GUID_0519358C_2F66_032D_63C6_2BC545D0AFB4'}
	(* Apply an inversion of the y-axis direction to an existing 2D affine transformation matrix. (expert function) *)
	FUNCTION F_VN_ApplyYAxisInversionToAffineTransformationExp : HRESULT
	VAR_INPUT
		aTransformationMatrix	:	REFERENCE TO TcVnMatrix2x3_LREAL;	(* Affine transformation matrix to which the inversion of the y-axis direction is applied *)
		bUsePreMultiplication	:	BOOL;	(* Select if pre- or post-multiplication should be used *)
		hrPrev	:	HRESULT;	(* HRESULT indicating the result of previous operations (If SUCCEEDED(hrPrev) equals false, no operation is executed.) *)
	END_VAR

END_FUNCTION

// Functions/Geometric and Coordinate Transformations/F_VN_ConvertCartesianToPolarAngleImage

	{attribute 'TcIecLibraryType'}
	{attribute 'external_name' := 'F_VN_ConvertCartesianToPolarAngleImage_GUID_17EADBBD_F562_070F_5C5C_9C9C6F0DA8B4'}
	(* Converts cartesian coordinates (x, y) to polar angle. *)
	FUNCTION F_VN_ConvertCartesianToPolarAngleImage : HRESULT
	VAR_INPUT
		ipSrcImageX	:	ITcVnImage;	(* Source image containing the x values (elements of type REAL or LREAL) *)
		ipSrcImageY	:	ITcVnImage;	(* Source image containing the y values (Same element type as ipSrcImageX) *)
		ipDestImageAng	:	REFERENCE TO ITcVnImage;	(* Destination image containing the angles (Same element type as source images. An appropriate destination image will be created if required.) *)
		hrPrev	:	HRESULT;	(* HRESULT indicating the result of previous operations (If SUCCEEDED(hrPrev) equals false, no operation is executed.) *)
	END_VAR

END_FUNCTION

// Functions/Geometric and Coordinate Transformations/F_VN_ConvertCartesianToPolarAngleImageExp

	{attribute 'TcIecLibraryType'}
	{attribute 'external_name' := 'F_VN_ConvertCartesianToPolarAngleImageExp_GUID_1D68747B_2AEF_02D8_5804_BAE8BD678C2F'}
	(* Converts cartesian coordinates (x, y) to polar angle. (expert function) *)
	FUNCTION F_VN_ConvertCartesianToPolarAngleImageExp : HRESULT
	VAR_INPUT
		ipSrcImageX	:	ITcVnImage;	(* Source image containing the x values (elements of type REAL or LREAL) *)
		ipSrcImageY	:	ITcVnImage;	(* Source image containing the y values (Same element type as ipSrcImageX) *)
		ipDestImageAng	:	REFERENCE TO ITcVnImage;	(* Destination image containing the angles (Same element type as source images. An appropriate destination image will be created if required.) *)
		bAngleInDegrees	:	BOOL;	(* Specifys, if the angles should be in degrees or radians *)
		hrPrev	:	HRESULT;	(* HRESULT indicating the result of previous operations (If SUCCEEDED(hrPrev) equals false, no operation is executed.) *)
	END_VAR

END_FUNCTION

// Functions/Geometric and Coordinate Transformations/F_VN_ConvertCartesianToPolarAngles

	{attribute 'TcIecLibraryType'}
	{attribute 'external_name' := 'F_VN_ConvertCartesianToPolarAngles_GUID_E7144BB7_132A_0642_64B6_73DCB69099EE'}
	(* Converts cartesian coordinates (x, y) to polar angle. *)
	FUNCTION F_VN_ConvertCartesianToPolarAngles : HRESULT
	VAR_INPUT
		ipSrcPointsCart	:	ITcVnContainer;	(* Container with cartesian points (ContainerType_Vector_TcVnPoint2_DINT or ContainerType_Vector_TcVnPoint2_REAL or ContainerType_Vector_TcVnPoint2_LREAL) *)
		ipDestAngles	:	REFERENCE TO ITcVnContainer;	(* Returns a container which is filled with the angles (ContainerType_Vector_REAL, if source points are of type TcVnPoint2_DINT or TcVnPoint2_REAL; else ContainerType_Vector_LREAL. Non-zero interface pointers are reused.) *)
		hrPrev	:	HRESULT;	(* HRESULT indicating the result of previous operations (If SUCCEEDED(hrPrev) equals false, no operation is executed.) *)
	END_VAR

END_FUNCTION

// Functions/Geometric and Coordinate Transformations/F_VN_ConvertCartesianToPolarAnglesExp

	{attribute 'TcIecLibraryType'}
	{attribute 'external_name' := 'F_VN_ConvertCartesianToPolarAnglesExp_GUID_5114B8BE_DDFA_0141_6749_A3EDE6F2388B'}
	(* Converts cartesian coordinates (x, y) to polar angle. (expert function) *)
	FUNCTION F_VN_ConvertCartesianToPolarAnglesExp : HRESULT
	VAR_INPUT
		ipSrcPointsCart	:	ITcVnContainer;	(* Container with cartesian points (ContainerType_Vector_TcVnPoint2_DINT or ContainerType_Vector_TcVnPoint2_REAL or ContainerType_Vector_TcVnPoint2_LREAL) *)
		ipDestAngles	:	REFERENCE TO ITcVnContainer;	(* Returns a container which is filled with the angles (ContainerType_Vector_REAL, if source points are of type TcVnPoint2_DINT or TcVnPoint2_REAL; else ContainerType_Vector_LREAL. Non-zero interface pointers are reused.) *)
		bAngleInDegrees	:	BOOL;	(* Specify, if the angles should be in degrees or radians *)
		hrPrev	:	HRESULT;	(* HRESULT indicating the result of previous operations (If SUCCEEDED(hrPrev) equals false, no operation is executed.) *)
	END_VAR

END_FUNCTION

// Functions/Geometric and Coordinate Transformations/F_VN_ConvertCartesianToPolarImages

	{attribute 'TcIecLibraryType'}
	{attribute 'external_name' := 'F_VN_ConvertCartesianToPolarImages_GUID_F8BA0872_BC93_0005_5BBA_C12C416537B0'}
	(* Converts cartesian coordinates (x, y) to polar coordinates (magnitude, angle). *)
	FUNCTION F_VN_ConvertCartesianToPolarImages : HRESULT
	VAR_INPUT
		ipSrcImageX	:	ITcVnImage;	(* Source image containing the x values (elements of type REAL or LREAL) *)
		ipSrcImageY	:	ITcVnImage;	(* Source image containing the y values (Same element type as ipSrcImageX) *)
		ipDestImageMag	:	REFERENCE TO ITcVnImage;	(* Destination image containing the magnitudes (Same element type as source images. An appropriate destination image will be created if required.) *)
		ipDestImageAng	:	REFERENCE TO ITcVnImage;	(* Destination image containing the angles (Same element type as source images. An appropriate destination image will be created if required.) *)
		hrPrev	:	HRESULT;	(* HRESULT indicating the result of previous operations (If SUCCEEDED(hrPrev) equals false, no operation is executed.) *)
	END_VAR

END_FUNCTION

// Functions/Geometric and Coordinate Transformations/F_VN_ConvertCartesianToPolarImagesExp

	{attribute 'TcIecLibraryType'}
	{attribute 'external_name' := 'F_VN_ConvertCartesianToPolarImagesExp_GUID_C7CB6E2F_D7A7_01AA_4CF2_0CB9BEF7AE79'}
	(* Converts cartesian coordinates (x, y) to polar coordinates (magnitude, angle). (expert function) *)
	FUNCTION F_VN_ConvertCartesianToPolarImagesExp : HRESULT
	VAR_INPUT
		ipSrcImageX	:	ITcVnImage;	(* Source image containing the x values (elements of type REAL or LREAL) *)
		ipSrcImageY	:	ITcVnImage;	(* Source image containing the y values (Same element type as ipSrcImageX) *)
		ipDestImageMag	:	REFERENCE TO ITcVnImage;	(* Destination image containing the magnitudes (Same element type as source images. An appropriate destination image will be created if required.) *)
		ipDestImageAng	:	REFERENCE TO ITcVnImage;	(* Destination image containing the angles (Same element type as source images. An appropriate destination image will be created if required.) *)
		bAngleInDegrees	:	BOOL;	(* Specifys, if the angles should be in degrees or radians *)
		hrPrev	:	HRESULT;	(* HRESULT indicating the result of previous operations (If SUCCEEDED(hrPrev) equals false, no operation is executed.) *)
	END_VAR

END_FUNCTION

// Functions/Geometric and Coordinate Transformations/F_VN_ConvertCartesianToPolarMagnitudeImage

	{attribute 'TcIecLibraryType'}
	{attribute 'external_name' := 'F_VN_ConvertCartesianToPolarMagnitudeImage_GUID_0980D42D_B8E3_0140_5BED_CD7062AAA1CE'}
	(* Converts cartesian coordinates (x, y) to polar magnitude. *)
	FUNCTION F_VN_ConvertCartesianToPolarMagnitudeImage : HRESULT
	VAR_INPUT
		ipSrcImageX	:	ITcVnImage;	(* Source image containing the x values (elements of type REAL or LREAL) *)
		ipSrcImageY	:	ITcVnImage;	(* Source image containing the y values (Same element type as ipSrcImageX) *)
		ipDestImageMag	:	REFERENCE TO ITcVnImage;	(* Destination image containing the magnitudes (Same element type as source images. An appropriate destination image will be created if required.) *)
		hrPrev	:	HRESULT;	(* HRESULT indicating the result of previous operations (If SUCCEEDED(hrPrev) equals false, no operation is executed.) *)
	END_VAR

END_FUNCTION

// Functions/Geometric and Coordinate Transformations/F_VN_ConvertCartesianToPolarMagnitudes

	{attribute 'TcIecLibraryType'}
	{attribute 'external_name' := 'F_VN_ConvertCartesianToPolarMagnitudes_GUID_173857FF_4E6E_0CA7_5502_B75DD11834D0'}
	(* Converts cartesian coordinates (x, y) to polar magnitude. *)
	FUNCTION F_VN_ConvertCartesianToPolarMagnitudes : HRESULT
	VAR_INPUT
		ipSrcPointsCart	:	ITcVnContainer;	(* Container with cartesian points (ContainerType_Vector_TcVnPoint2_DINT or ContainerType_Vector_TcVnPoint2_REAL or ContainerType_Vector_TcVnPoint2_LREAL) *)
		ipDestMags	:	REFERENCE TO ITcVnContainer;	(* Returns a container which is filled with the magnitudes (ContainerType_Vector_REAL, if source points are of type TcVnPoint2_DINT or TcVnPoint2_REAL; else ContainerType_Vector_LREAL. Non-zero interface pointers are reused.) *)
		hrPrev	:	HRESULT;	(* HRESULT indicating the result of previous operations (If SUCCEEDED(hrPrev) equals false, no operation is executed.) *)
	END_VAR

END_FUNCTION

// Functions/Geometric and Coordinate Transformations/F_VN_ConvertCartesianToPolarPoints

	{attribute 'TcIecLibraryType'}
	{attribute 'external_name' := 'F_VN_ConvertCartesianToPolarPoints_GUID_1B7EE36C_3385_0761_6D0F_583B6ACA8374'}
	(* Converts cartesian coordinates (x, y) to polar coordinates (magnitude, angle). *)
	FUNCTION F_VN_ConvertCartesianToPolarPoints : HRESULT
	VAR_INPUT
		ipSrcPointsCart	:	ITcVnContainer;	(* Container with cartesian points (ContainerType_Vector_TcVnPoint2_DINT or ContainerType_Vector_TcVnPoint2_REAL or ContainerType_Vector_TcVnPoint2_LREAL) *)
		ipDestPointsPolar	:	REFERENCE TO ITcVnContainer;	(* Returns a container which is filled with the converted points in polar coordinates (ContainerType_Vector_TcVnPoint2_REAL, if source points are of type TcVnPoint2_DINT or TcVnPoint2_REAL; else ContainerType_Vector_TcVnPoint2_LREAL. Non-zero interface pointers are reused.) *)
		hrPrev	:	HRESULT;	(* HRESULT indicating the result of previous operations (If SUCCEEDED(hrPrev) equals false, no operation is executed.) *)
	END_VAR

END_FUNCTION

// Functions/Geometric and Coordinate Transformations/F_VN_ConvertCartesianToPolarPointsExp

	{attribute 'TcIecLibraryType'}
	{attribute 'external_name' := 'F_VN_ConvertCartesianToPolarPointsExp_GUID_7BD14587_5533_0AF9_4CDD_1791B980D155'}
	(* Converts cartesian coordinates (x, y) to polar coordinates (magnitude, angle). (expert function) *)
	FUNCTION F_VN_ConvertCartesianToPolarPointsExp : HRESULT
	VAR_INPUT
		ipSrcPointsCart	:	ITcVnContainer;	(* Container with cartesian points (ContainerType_Vector_TcVnPoint2_DINT or ContainerType_Vector_TcVnPoint2_REAL or ContainerType_Vector_TcVnPoint2_LREAL) *)
		ipDestPointsPolar	:	REFERENCE TO ITcVnContainer;	(* Returns a container which is filled with the converted points in polar coordinates (ContainerType_Vector_TcVnPoint2_REAL, if source points are of type TcVnPoint2_DINT or TcVnPoint2_REAL; else ContainerType_Vector_TcVnPoint2_LREAL. Non-zero interface pointers are reused.) *)
		bAngleInDegrees	:	BOOL;	(* Specifys, if the angles should be in degrees or radians *)
		hrPrev	:	HRESULT;	(* HRESULT indicating the result of previous operations (If SUCCEEDED(hrPrev) equals false, no operation is executed.) *)
	END_VAR

END_FUNCTION

// Functions/Geometric and Coordinate Transformations/F_VN_ConvertPolarToCartesianImages

	{attribute 'TcIecLibraryType'}
	{attribute 'external_name' := 'F_VN_ConvertPolarToCartesianImages_GUID_D58D94D9_F6D8_04ED_4732_1550D7DAAC18'}
	(* Converts polar coordinates (magnitude, angle) to cartesian coordinates (x, y). *)
	FUNCTION F_VN_ConvertPolarToCartesianImages : HRESULT
	VAR_INPUT
		ipSrcImageMag	:	ITcVnImage;	(* Source image containing the magnitudes (elements of type REAL or LREAL) *)
		ipSrcImageAng	:	ITcVnImage;	(* Source image containing the angles (Same element type as ipSrcImageMag) *)
		ipDestImageX	:	REFERENCE TO ITcVnImage;	(* Destination image containing the x values (Same element type as source images. An appropriate destination image will be created if required.) *)
		ipDestImageY	:	REFERENCE TO ITcVnImage;	(* Destination image containing the y values (Same element type as source images. An appropriate destination image will be created if required.) *)
		hrPrev	:	HRESULT;	(* HRESULT indicating the result of previous operations (If SUCCEEDED(hrPrev) equals false, no operation is executed.) *)
	END_VAR

END_FUNCTION

// Functions/Geometric and Coordinate Transformations/F_VN_ConvertPolarToCartesianImagesExp

	{attribute 'TcIecLibraryType'}
	{attribute 'external_name' := 'F_VN_ConvertPolarToCartesianImagesExp_GUID_8ADAC3A5_4456_0FD2_7554_A61782C6C355'}
	(* Converts polar coordinates (magnitude, angle) to cartesian coordinates (x, y). (expert function) *)
	FUNCTION F_VN_ConvertPolarToCartesianImagesExp : HRESULT
	VAR_INPUT
		ipSrcImageMag	:	ITcVnImage;	(* Source image containing the magnitudes (elements of type REAL or LREAL) *)
		ipSrcImageAng	:	ITcVnImage;	(* Source image containing the angles (Same element type as ipSrcImageMag) *)
		ipDestImageX	:	REFERENCE TO ITcVnImage;	(* Destination image containing the x values (Same element type as source images. An appropriate destination image will be created if required.) *)
		ipDestImageY	:	REFERENCE TO ITcVnImage;	(* Destination image containing the y values (Same element type as source images. An appropriate destination image will be created if required.) *)
		bAngleInDegrees	:	BOOL;	(* Specifys, if the angles are in degrees or radians *)
		hrPrev	:	HRESULT;	(* HRESULT indicating the result of previous operations (If SUCCEEDED(hrPrev) equals false, no operation is executed.) *)
	END_VAR

END_FUNCTION

// Functions/Geometric and Coordinate Transformations/F_VN_ConvertPolarToCartesianPoints

	{attribute 'TcIecLibraryType'}
	{attribute 'external_name' := 'F_VN_ConvertPolarToCartesianPoints_GUID_5DF61BFC_CDA0_0EA0_706A_507F6E239E48'}
	(* Converts polar coordinates (magnitude, angle) to cartesian coordinates (x, y). *)
	FUNCTION F_VN_ConvertPolarToCartesianPoints : HRESULT
	VAR_INPUT
		ipSrcPointsPolar	:	ITcVnContainer;	(* Container with polar coordinates (ContainerType_Vector_TcVnPoint2_REAL or ContainerType_Vector_TcVnPoint2_LREAL) *)
		ipDestPointsCart	:	REFERENCE TO ITcVnContainer;	(* Returns a container which is filled with the converted points in cartesian coordinates (same type ID as ipSrcPointsPolar. Non-zero interface pointers are reused.) *)
		hrPrev	:	HRESULT;	(* HRESULT indicating the result of previous operations (If SUCCEEDED(hrPrev) equals false, no operation is executed.) *)
	END_VAR

END_FUNCTION

// Functions/Geometric and Coordinate Transformations/F_VN_ConvertPolarToCartesianPointsExp

	{attribute 'TcIecLibraryType'}
	{attribute 'external_name' := 'F_VN_ConvertPolarToCartesianPointsExp_GUID_01E044CB_F7C3_0F9D_7A9D_DCCA17D89581'}
	(* Converts polar coordinates (magnitude, angle) to cartesian coordinates (x, y). (expert function) *)
	FUNCTION F_VN_ConvertPolarToCartesianPointsExp : HRESULT
	VAR_INPUT
		ipSrcPointsPolar	:	ITcVnContainer;	(* Container with polar coordinates (ContainerType_Vector_TcVnPoint2_REAL or ContainerType_Vector_TcVnPoint2_LREAL) *)
		ipDestPointsCart	:	REFERENCE TO ITcVnContainer;	(* Returns a container which is filled with the converted points in cartesian coordinates (same type ID as ipSrcPointsPolar. Non-zero interface pointers are reused.) *)
		bAngleInDegrees	:	BOOL;	(* Specifys, if the angles are in degrees or radians *)
		hrPrev	:	HRESULT;	(* HRESULT indicating the result of previous operations (If SUCCEEDED(hrPrev) equals false, no operation is executed.) *)
	END_VAR

END_FUNCTION

// Functions/Geometric and Coordinate Transformations/F_VN_DecomposeAffineTransformation

	{attribute 'TcIecLibraryType'}
	{attribute 'external_name' := 'F_VN_DecomposeAffineTransformation_GUID_08BAC7AF_F12F_0114_702C_9D677E9A3BF3'}
	(* Decompose an affine transformation matrix and return the rotation angle (clockwise) in radian. The decomposition method assumes the following order of transformation: Translation, Rotation, Scale, and Skew. *)
	FUNCTION F_VN_DecomposeAffineTransformation : HRESULT
	VAR_INPUT
		aAffineTransform	:	REFERENCE TO TcVnMatrix2x3_LREAL;	(* Affine transformation matrix *)
		fRotationAngle	:	REFERENCE TO LREAL;	(* Rotation angle (radian) in the clockwise direction. The rotation center is the origin point (0,0) *)
		hrPrev	:	HRESULT;	(* HRESULT indicating the result of previous operations (If SUCCEEDED(hrPrev) equals false, no operation is executed.) *)
	END_VAR

END_FUNCTION

// Functions/Geometric and Coordinate Transformations/F_VN_DecomposeAffineTransformationExp

	{attribute 'TcIecLibraryType'}
	{attribute 'external_name' := 'F_VN_DecomposeAffineTransformationExp_GUID_0A19BB33_E82A_0D97_5DAF_4E324AD68E62'}
	(* Decompose an affine transformation matrix and return the rotation angle (clockwise) in radian, translation vector (pixels), scale, and skew vectors (angle in radian). The decomposition method assumes the following order of transformation: Translation, Rotation, Scale, and Skew. *)
	FUNCTION F_VN_DecomposeAffineTransformationExp : HRESULT
	VAR_INPUT
		aAffineTransform	:	REFERENCE TO TcVnMatrix2x3_LREAL;	(* Affine transformation matrix *)
		fRotationAngle	:	REFERENCE TO LREAL;	(* Rotation angle (radian) in the clockwise direction. The rotation center is the origin point (0,0) *)
		aTranslationVector	:	REFERENCE TO TcVnVector2_LREAL;	(* 2D translation vector. The values are in pixels *)
		aScaleVector	:	REFERENCE TO TcVnVector2_LREAL;	(* 2D scale vector  *)
		aSkewVector	:	REFERENCE TO TcVnVector2_LREAL;	(* 2D skew vector. The values are the skew angles in x and y directions in radian *)
		hrPrev	:	HRESULT;	(* HRESULT indicating the result of previous operations (If SUCCEEDED(hrPrev) equals false, no operation is executed.) *)
	END_VAR

END_FUNCTION

// Functions/Geometric and Coordinate Transformations/F_VN_DecomposeHomography

	{attribute 'TcIecLibraryType'}
	{attribute 'external_name' := 'F_VN_DecomposeHomography_GUID_089F1EA7_6A4F_0D6C_5E68_EBEB6EEB5CD0'}
	(* Decompose a homography matrix into four solutions of rotation, translation, and plane normal. It returns two solutions (Ra, Ta, Nb) and (Rb, Tb, Nb). The third and the fourth solutions can be calculated as follows: (Ra, -Ta, -Na) and (Rb, -Tb, -Nb). *)
	FUNCTION F_VN_DecomposeHomography : HRESULT
	VAR_INPUT
		aHomography	:	REFERENCE TO TcVnMatrix3x3_LREAL;	(* Homography matrix (a perspective transformation between two planes) *)
		aCameraMatrix	:	REFERENCE TO TcVnMatrix3x3_LREAL;	(* Camera matrix *)
		aRotationMatrixA	:	REFERENCE TO TcVnMatrix3x3_LREAL;	(* Rotation matrix of the first solution (Ra) *)
		aTranslationVectorA	:	REFERENCE TO TcVnVector3_LREAL;	(* Translation vector of the first solution (Ta) *)
		aNormVectorA	:	REFERENCE TO TcVnVector3_LREAL;	(* Norm vector of the first solution (Na) *)
		aRotationMatrixB	:	REFERENCE TO TcVnMatrix3x3_LREAL;	(* Rotation matrix of the second solution (Rb) *)
		aTranslationVectorB	:	REFERENCE TO TcVnVector3_LREAL;	(* Translation vector of the second solution (Tb) *)
		aNormVectorB	:	REFERENCE TO TcVnVector3_LREAL;	(* Norm vector of the second solution Nb *)
		hrPrev	:	HRESULT;	(* HRESULT indicating the result of previous operations (If SUCCEEDED(hrPrev) equals false, no operation is executed.) *)
	END_VAR
	VAR_OUTPUT
		nSolutions	:	UDINT;	(* Returns the number of solutions. In normal cases, it is equal four.  *)
	END_VAR

END_FUNCTION

// Functions/Geometric and Coordinate Transformations/F_VN_DecomposeHomographyExp

	{attribute 'TcIecLibraryType'}
	{attribute 'external_name' := 'F_VN_DecomposeHomographyExp_GUID_743C436F_8617_0168_5F3C_08312E89C57E'}
	(* Decompose a homography matrix and verify four solutions of rotation, translation, and plane normal. It uses visible reference points being in front of the camera to confirm which solution(s) of the four solutions (maximum two solutions) are consistent with all reference points. *)
	FUNCTION F_VN_DecomposeHomographyExp : HRESULT
	VAR_INPUT
		aHomography	:	REFERENCE TO TcVnMatrix3x3_LREAL;	(* Homography matrix (a perspective transformation between two planes) *)
		aCameraMatrix	:	REFERENCE TO TcVnMatrix3x3_LREAL;	(* Camera matrix *)
		aRotationMatrixA	:	REFERENCE TO TcVnMatrix3x3_LREAL;	(* Rotation matrix of the first solution (Ra) *)
		aTranslationVectorA	:	REFERENCE TO TcVnVector3_LREAL;	(* Translation vector of the first solution (Ta) *)
		aNormVectorA	:	REFERENCE TO TcVnVector3_LREAL;	(* Norm vector of the first solution (Na) *)
		aRotationMatrixB	:	REFERENCE TO TcVnMatrix3x3_LREAL;	(* Rotation matrix of the second solution (Rb) *)
		aTranslationVectorB	:	REFERENCE TO TcVnVector3_LREAL;	(* Translation vector of the second solution (Tb) *)
		aNormVectorB	:	REFERENCE TO TcVnVector3_LREAL;	(* Norm vector of the second solution (Nb) *)
		ipPointsSrc	:	ITcVnContainer;	(* Container with source points (ContainerType_Vector_TcVnPoint2_REAL) *)
		ipPointsDes	:	ITcVnContainer;	(* Container with destination points (same number as ipPoints1, ContainerType_Vector_TcVnPoint2_REAL) *)
		ipInlierMask	:	ITcVnContainer;	(* A mask marking the inliers (optional, set to 0 if not available; ContainerType_Vector_SINT or ContainerType_Vector_USINT) *)
		hrPrev	:	HRESULT;	(* HRESULT indicating the result of previous operations (If SUCCEEDED(hrPrev) equals false, no operation is executed.) *)
	END_VAR
	VAR_OUTPUT
		nSolutions	:	UDINT;	(* Return the number of true potential solutions [0,1, or 2].
							0: no true potential solutions for the given corresponding points are confirmed.
							1: the solution (Ra, Ta, Na) is confirmed.
							2: both solution (Ra, Ta, Na) and (Rb, Tb, Nb) are confirmed.
							In all cases the function returns two solutions (Ra, Ta, Nb) and (Rb, Tb, Nb). The third and the fourth solutions can be calculated as follows: (Ra, -Ta, -Na) and (Rb, -Tb, -Nb).
						 *)
	END_VAR

END_FUNCTION

// Functions/Geometric and Coordinate Transformations/F_VN_FlipImage

	{attribute 'TcIecLibraryType'}
	{attribute 'external_name' := 'F_VN_FlipImage_GUID_D8DC2A9F_113D_0952_5EA3_CC03711333D7'}
	(* Flip an image (mirror and shift back to prior coordinates). *)
	FUNCTION F_VN_FlipImage : HRESULT
	VAR_INPUT
		ipSrcImage	:	ITcVnImage;	(* Source image *)
		ipDestImage	:	REFERENCE TO ITcVnImage;	(* Destination image (An appropriate destination image will be created if required.) *)
		eFlipAxis	:	ETcVnFlipAxis;	(* Selects the axis around which to flip the image *)
		hrPrev	:	HRESULT;	(* HRESULT indicating the result of previous operations (If SUCCEEDED(hrPrev) equals false, no operation is executed.) *)
	END_VAR

END_FUNCTION

// Functions/Geometric and Coordinate Transformations/F_VN_GenerateAffineTransformationUnitMatrix2D

	{attribute 'TcIecLibraryType'}
	{attribute 'external_name' := 'F_VN_GenerateAffineTransformationUnitMatrix2D_GUID_9E1964AA_3221_0763_59D5_5D98A3F99DCD'}
	(* Generate an affine transformation 2D unit matrix. *)
	FUNCTION F_VN_GenerateAffineTransformationUnitMatrix2D : HRESULT
	VAR_INPUT
		aTransformationMatrix	:	REFERENCE TO TcVnMatrix2x3_LREAL;	(* Resulting affine transformation unit matrix *)
		hrPrev	:	HRESULT;	(* HRESULT indicating the result of previous operations (If SUCCEEDED(hrPrev) equals false, no operation is executed.) *)
	END_VAR

END_FUNCTION

// Functions/Geometric and Coordinate Transformations/F_VN_GetAffineTransformation

	{attribute 'TcIecLibraryType'}
	{attribute 'external_name' := 'F_VN_GetAffineTransformation_GUID_EFFB7141_B734_03CC_5DA4_F78600A68161'}
	(* Calculate the affine transformation between three corresponding point pairs. The points mark the corners of the corresponding triangles. *)
	FUNCTION F_VN_GetAffineTransformation : HRESULT
	VAR_INPUT
		aSrcPoints	:	REFERENCE TO TcVnArray3_Point2_REAL;	(* Source points *)
		aDestPoints	:	REFERENCE TO TcVnArray3_Point2_REAL;	(* Destination points *)
		aTransformationMatrix	:	REFERENCE TO TcVnMatrix2x3_LREAL;	(* Resulting transformation matrix *)
		hrPrev	:	HRESULT;	(* HRESULT indicating the result of previous operations (If SUCCEEDED(hrPrev) equals false, no operation is executed.) *)
	END_VAR

END_FUNCTION

// Functions/Geometric and Coordinate Transformations/F_VN_GetAffineTransformation2D

	{attribute 'TcIecLibraryType'}
	{attribute 'external_name' := 'F_VN_GetAffineTransformation2D_GUID_E5A0B378_38E7_0A58_53F9_5224B7730F7D'}
	(* Estimate the 2D affine transformation between two planar point sets using RANSAC algorithm. *)
	FUNCTION F_VN_GetAffineTransformation2D : HRESULT
	VAR_INPUT
		ipSrcPoints	:	ITcVnContainer;	(* Container with at least 3 source points (ContainerType_Vector_TcVnPoint2_REAL) *)
		ipDestPoints	:	ITcVnContainer;	(* Container with destination points (same number as ipSrcPoints, ContainerType_Vector_TcVnPoint2_REAL) *)
		aAffineTransform	:	REFERENCE TO TcVnMatrix2x3_LREAL;	(* Returns the affine transformation matrix, which transforms the source points to the destination points *)
		hrPrev	:	HRESULT;	(* HRESULT indicating the result of previous operations (If SUCCEEDED(hrPrev) equals false, no operation is executed.) *)
	END_VAR

END_FUNCTION

// Functions/Geometric and Coordinate Transformations/F_VN_GetAffineTransformation2DExp

	{attribute 'TcIecLibraryType'}
	{attribute 'external_name' := 'F_VN_GetAffineTransformation2DExp_GUID_3741B428_3322_0947_5DEA_A716F72BD0FE'}
	(* Estimate the affine transformation between two planar point sets. (expert function) *)
	FUNCTION F_VN_GetAffineTransformation2DExp : HRESULT
	VAR_INPUT
		ipSrcPoints	:	ITcVnContainer;	(* Container with at least 3 source points (ContainerType_Vector_TcVnPoint2_REAL) *)
		ipDestPoints	:	ITcVnContainer;	(* Container with destination points (same number as ipSrcPoints, ContainerType_Vector_TcVnPoint2_REAL) *)
		aAffineTransform	:	REFERENCE TO TcVnMatrix2x3_LREAL;	(* Returns the affine transformation matrix, which transforms the source points to the destination points *)
		eAlgorithm	:	ETcVnEstimationAlgorithm;	(* Estimation algorithm (only RANSAC and LMEDS are supported) *)
		fReprojThreshold	:	LREAL;	(* Maximum allowed reprojection error to treat a point pair as an inlier *)
		ipInlierMask	:	REFERENCE TO ITcVnContainer;	(* Returns a mask marking the inliers (optional, set to 0 if not required; ContainerType_Vector_USINT) *)
		nMaxIterations	:	UDINT;	(* Maximum number of iterations *)
		fConfidence	:	LREAL;	(* Confidence (0..1) *)
		nRefineIters	:	UDINT;	(* Maximum number of iterations of Levenberg-Marquardt algorithm to refine further the affine transform (using only inliers). Set to 0 to disable refining. *)
		hrPrev	:	HRESULT;	(* HRESULT indicating the result of previous operations (If SUCCEEDED(hrPrev) equals false, no operation is executed.) *)
	END_VAR

END_FUNCTION

// Functions/Geometric and Coordinate Transformations/F_VN_GetPerspectiveTransformation

	{attribute 'TcIecLibraryType'}
	{attribute 'external_name' := 'F_VN_GetPerspectiveTransformation_GUID_63152C06_C780_03DB_7A40_23A2047B16AC'}
	(* Calculate the perspective transformation between four corresponding point pairs. The points mark the corners of the corresponding rectangles. *)
	FUNCTION F_VN_GetPerspectiveTransformation : HRESULT
	VAR_INPUT
		aSrcPoints	:	REFERENCE TO TcVnArray4_Point2_REAL;	(* Source points *)
		aDestPoints	:	REFERENCE TO TcVnArray4_Point2_REAL;	(* Destination points *)
		aTransformationMatrix	:	REFERENCE TO TcVnMatrix3x3_LREAL;	(* Resulting transformation matrix *)
		hrPrev	:	HRESULT;	(* HRESULT indicating the result of previous operations (If SUCCEEDED(hrPrev) equals false, no operation is executed.) *)
	END_VAR

END_FUNCTION

// Functions/Geometric and Coordinate Transformations/F_VN_Homography

	{attribute 'TcIecLibraryType'}
	{attribute 'external_name' := 'F_VN_Homography_GUID_1DD54F52_FEE1_0DBB_4A2E_95C87BF73F63'}
	(* Find the homography (perspective transformation) between two planar point sets using RANSAC algorithm. *)
	FUNCTION F_VN_Homography : HRESULT
	VAR_INPUT
		ipSrcPoints	:	ITcVnContainer;	(* Container with at least 4 source points (ContainerType_Vector_TcVnPoint2_REAL) *)
		ipDestPoints	:	ITcVnContainer;	(* Container with destination points (same number as ipSrcPoints, ContainerType_Vector_TcVnPoint2_REAL) *)
		aPerspectiveTransform	:	REFERENCE TO TcVnMatrix3x3_LREAL;	(* Returns the perspective transformation matrix, which transforms the source points to the destination points *)
		hrPrev	:	HRESULT;	(* HRESULT indicating the result of previous operations (If SUCCEEDED(hrPrev) equals false, no operation is executed.) *)
	END_VAR

END_FUNCTION

// Functions/Geometric and Coordinate Transformations/F_VN_HomographyExp

	{attribute 'TcIecLibraryType'}
	{attribute 'external_name' := 'F_VN_HomographyExp_GUID_326059F8_2999_0C79_755C_D1EC7D873134'}
	(* Find the homography (perspective transformation) between two planar point sets. (expert function) *)
	FUNCTION F_VN_HomographyExp : HRESULT
	VAR_INPUT
		ipSrcPoints	:	ITcVnContainer;	(* Container with at least 4 source points (ContainerType_Vector_TcVnPoint2_REAL) *)
		ipDestPoints	:	ITcVnContainer;	(* Container with destination points (same number as ipSrcPoints, ContainerType_Vector_TcVnPoint2_REAL) *)
		aPerspectiveTransform	:	REFERENCE TO TcVnMatrix3x3_LREAL;	(* Returns the perspective transformation matrix, which transforms the source points to the destination points *)
		eAlgorithm	:	ETcVnEstimationAlgorithm;	(* Estimation algorithm *)
		fReprojThreshold	:	LREAL;	(* Maximum allowed reprojection error to treat a point pair as an inlier (only for RANSAC, RHO) *)
		ipInlierMask	:	REFERENCE TO ITcVnContainer;	(* Returns a mask marking the inliers (optional, set to 0 if not required; ContainerType_Vector_SINT; only for RANSAC, LMEDS) *)
		nMaxIterations	:	UDINT;	(* Maximum number of RANSAC iterations *)
		fConfidence	:	LREAL;	(* Confidence (0..1) *)
		hrPrev	:	HRESULT;	(* HRESULT indicating the result of previous operations (If SUCCEEDED(hrPrev) equals false, no operation is executed.) *)
	END_VAR

END_FUNCTION

// Functions/Geometric and Coordinate Transformations/F_VN_InvertAffineTransformation

	{attribute 'TcIecLibraryType'}
	{attribute 'external_name' := 'F_VN_InvertAffineTransformation_GUID_3BC8AD5D_FF69_05C1_7A08_9668B3671CBB'}
	(* Invert a 2D affine transformation matrix. The inverted transformation compensates the affine transformation on an image if it is used in the F_VN_WarpAffine function. *)
	FUNCTION F_VN_InvertAffineTransformation : HRESULT
	VAR_INPUT
		aTransformationMatrix	:	REFERENCE TO TcVnMatrix2x3_LREAL;	(* Source affine transformation matrix *)
		aInvertedTransformationMatrix	:	REFERENCE TO TcVnMatrix2x3_LREAL;	(* Resulting inverted affine transformation matrix *)
		hrPrev	:	HRESULT;	(* HRESULT indicating the result of previous operations (If SUCCEEDED(hrPrev) equals false, no operation is executed.) *)
	END_VAR

END_FUNCTION

// Functions/Geometric and Coordinate Transformations/F_VN_WarpAffine

	{attribute 'TcIecLibraryType'}
	{attribute 'external_name' := 'F_VN_WarpAffine_GUID_801D8F20_1812_01A0_5AB3_7739626B998B'}
	(* Apply an affine transformation to an image. *)
	FUNCTION F_VN_WarpAffine : HRESULT
	VAR_INPUT
		ipSrcImage	:	ITcVnImage;	(* Source image *)
		ipDestImage	:	REFERENCE TO ITcVnImage;	(* Destination image (An appropriate image will be created if required.) *)
		aTransformationMatrix	:	REFERENCE TO TcVnMatrix2x3_LREAL;	(* Affine transformation matrix *)
		hrPrev	:	HRESULT;	(* HRESULT indicating the result of previous operations (If SUCCEEDED(hrPrev) equals false, no operation is executed.) *)
	END_VAR

END_FUNCTION

// Functions/Geometric and Coordinate Transformations/F_VN_PerspectiveTransformation

	{attribute 'TcIecLibraryType'}
	{attribute 'external_name' := 'F_VN_PerspectiveTransformation_GUID_0610B54F_6BF6_0DF4_7696_7DF5159B3287'}
	(* Apply a perspective transformation (rotation + translation, e.g. from extrinsic calibration) to 3D point coordinates. *)
	FUNCTION F_VN_PerspectiveTransformation : HRESULT
	VAR_INPUT
		ipSrcPoints	:	ITcVnContainer;	(* Container with 3D source points (TcVnPoint3_REAL or TcVnPoint3_LREAL) *)
		ipDestPoints	:	REFERENCE TO ITcVnContainer;	(* Returns the transformed points (same type as ipSrcPoints) *)
		aRotationMatrix	:	REFERENCE TO TcVnMatrix3x3_LREAL;	(* 3x3 rotation matrix *)
		aTranslationVector	:	REFERENCE TO TcVnVector3_LREAL;	(* Translation vector *)
		hrPrev	:	HRESULT;	(* HRESULT indicating the result of previous operations (If SUCCEEDED(hrPrev) equals false, no operation is executed.) *)
	END_VAR

END_FUNCTION

// Functions/Geometric and Coordinate Transformations/F_VN_PyramidDown

	{attribute 'TcIecLibraryType'}
	{attribute 'external_name' := 'F_VN_PyramidDown_GUID_037757AD_A7A8_0F3B_6BF2_5CAF407EBB48'}
	(* Downsamples an image to half width and height. *)
	FUNCTION F_VN_PyramidDown : HRESULT
	VAR_INPUT
		ipSrcImage	:	ITcVnImage;	(* Source image *)
		ipDestImage	:	REFERENCE TO ITcVnImage;	(* Destination image (An appropriate destination image will be created if required.) *)
		hrPrev	:	HRESULT;	(* HRESULT indicating the result of previous operations (If SUCCEEDED(hrPrev) equals false, no operation is executed.) *)
	END_VAR

END_FUNCTION

// Functions/Geometric and Coordinate Transformations/F_VN_PyramidUp

	{attribute 'TcIecLibraryType'}
	{attribute 'external_name' := 'F_VN_PyramidUp_GUID_60795244_3FC4_095F_732B_EC2BF1571832'}
	(* Upsamples an image to double width and height. *)
	FUNCTION F_VN_PyramidUp : HRESULT
	VAR_INPUT
		ipSrcImage	:	ITcVnImage;	(* Source image *)
		ipDestImage	:	REFERENCE TO ITcVnImage;	(* Destination image (An appropriate destination image will be created if required.) *)
		hrPrev	:	HRESULT;	(* HRESULT indicating the result of previous operations (If SUCCEEDED(hrPrev) equals false, no operation is executed.) *)
	END_VAR

END_FUNCTION

// Functions/Geometric and Coordinate Transformations/F_VN_RemapImageToLogPolarSpace

	{attribute 'TcIecLibraryType'}
	{attribute 'external_name' := 'F_VN_RemapImageToLogPolarSpace_GUID_9665D1C5_1A95_088B_46EE_7AA704020B91'}
	(* Remap an image to log-polar space. *)
	FUNCTION F_VN_RemapImageToLogPolarSpace : HRESULT
	VAR_INPUT
		ipSrcImage	:	ITcVnImage;	(* Source image *)
		ipDestImage	:	REFERENCE TO ITcVnImage;	(* Destination image (Must not be the same as ipSrcImage! An appropriate destination image will be created if required.) *)
		aCenter	:	REFERENCE TO TcVnPoint2_REAL;	(* Center point for the transformation *)
		hrPrev	:	HRESULT;	(* HRESULT indicating the result of previous operations (If SUCCEEDED(hrPrev) equals false, no operation is executed.) *)
	END_VAR

END_FUNCTION

// Functions/Geometric and Coordinate Transformations/F_VN_RemapImageToLogPolarSpaceExp

	{attribute 'TcIecLibraryType'}
	{attribute 'external_name' := 'F_VN_RemapImageToLogPolarSpaceExp_GUID_6349A592_56D9_0AC0_703B_3960CE990A04'}
	(* Remap an image to log-polar space. (expert function) *)
	FUNCTION F_VN_RemapImageToLogPolarSpaceExp : HRESULT
	VAR_INPUT
		ipSrcImage	:	ITcVnImage;	(* Source image *)
		ipDestImage	:	REFERENCE TO ITcVnImage;	(* Destination image (Must not be the same as ipSrcImage! An appropriate destination image will be created if required.) *)
		aCenter	:	REFERENCE TO TcVnPoint2_REAL;	(* Center point for the transformation *)
		fScale	:	LREAL;	(* Magnitude scale parameter (set to 0 for auto select) *)
		eInterpolationType	:	ETcVnInterpolationType;	(* Interpolation type *)
		hrPrev	:	HRESULT;	(* HRESULT indicating the result of previous operations (If SUCCEEDED(hrPrev) equals false, no operation is executed.) *)
	END_VAR

END_FUNCTION

// Functions/Geometric and Coordinate Transformations/F_VN_RemapImageToPolarSpace

	{attribute 'TcIecLibraryType'}
	{attribute 'external_name' := 'F_VN_RemapImageToPolarSpace_GUID_26B9A858_1378_03D2_47F3_643E1B49D08F'}
	(* Remap an image to polar space. *)
	FUNCTION F_VN_RemapImageToPolarSpace : HRESULT
	VAR_INPUT
		ipSrcImage	:	ITcVnImage;	(* Source image *)
		ipDestImage	:	REFERENCE TO ITcVnImage;	(* Destination image (Must not be the same as ipSrcImage! An appropriate destination image will be created if required.) *)
		aCenter	:	REFERENCE TO TcVnPoint2_REAL;	(* Center point for the transformation *)
		hrPrev	:	HRESULT;	(* HRESULT indicating the result of previous operations (If SUCCEEDED(hrPrev) equals false, no operation is executed.) *)
	END_VAR

END_FUNCTION

// Functions/Geometric and Coordinate Transformations/F_VN_RemapImageToPolarSpaceExp

	{attribute 'TcIecLibraryType'}
	{attribute 'external_name' := 'F_VN_RemapImageToPolarSpaceExp_GUID_609CB515_4A4F_0AE6_5A28_7663ED9697A0'}
	(* Remap an image to polar space. (expert function) *)
	FUNCTION F_VN_RemapImageToPolarSpaceExp : HRESULT
	VAR_INPUT
		ipSrcImage	:	ITcVnImage;	(* Source image *)
		ipDestImage	:	REFERENCE TO ITcVnImage;	(* Destination image (Must not be the same as ipSrcImage! An appropriate destination image will be created if required.) *)
		aCenter	:	REFERENCE TO TcVnPoint2_REAL;	(* Center point for the transformation *)
		fMaxRadius	:	LREAL;	(* Maximum radius for the transformation (set to 0 for auto select) *)
		eInterpolationType	:	ETcVnInterpolationType;	(* Interpolation type *)
		hrPrev	:	HRESULT;	(* HRESULT indicating the result of previous operations (If SUCCEEDED(hrPrev) equals false, no operation is executed.) *)
	END_VAR

END_FUNCTION

// Functions/Geometric and Coordinate Transformations/F_VN_ResizeImage

	{attribute 'TcIecLibraryType'}
	{attribute 'external_name' := 'F_VN_ResizeImage_GUID_158C9B48_45C7_062C_78D6_262FF926E16D'}
	(* Resize an image using a specific interpolation type. *)
	FUNCTION F_VN_ResizeImage : HRESULT
	VAR_INPUT
		ipSrcImage	:	ITcVnImage;	(* Source image *)
		ipDestImage	:	REFERENCE TO ITcVnImage;	(* Destination image (An appropriate image will be created if required.) *)
		nWidth	:	UDINT;	(* New width *)
		nHeight	:	UDINT;	(* New height *)
		eInterpolationType	:	ETcVnInterpolationType;	(* Interpolation type *)
		hrPrev	:	HRESULT;	(* HRESULT indicating the result of previous operations (If SUCCEEDED(hrPrev) equals false, no operation is executed.) *)
	END_VAR

END_FUNCTION

// Functions/Geometric and Coordinate Transformations/F_VN_RotateImage

	{attribute 'TcIecLibraryType'}
	{attribute 'external_name' := 'F_VN_RotateImage_GUID_74576AFF_4EDD_060D_57EA_7896BA07C490'}
	(* Rotate an image by 90, 180, or 270 degrees in clockwise direction. *)
	FUNCTION F_VN_RotateImage : HRESULT
	VAR_INPUT
		ipSrcImage	:	ITcVnImage;	(* Source image *)
		ipDestImage	:	REFERENCE TO ITcVnImage;	(* Destination image (An appropriate image will be created if required.) *)
		eAngle	:	ETcVnRotationAngle;	(* Rotation angle *)
		hrPrev	:	HRESULT;	(* HRESULT indicating the result of previous operations (If SUCCEEDED(hrPrev) equals false, no operation is executed.) *)
	END_VAR

END_FUNCTION

// Functions/Geometric and Coordinate Transformations/F_VN_RotateImageExp

	{attribute 'TcIecLibraryType'}
	{attribute 'external_name' := 'F_VN_RotateImageExp_GUID_5ADC2A6C_CE4A_012F_6EA8_572FD65557CB'}
	(* Rotate an image by an individual rotation angle in degrees. *)
	FUNCTION F_VN_RotateImageExp : HRESULT
	VAR_INPUT
		ipSrcImage	:	ITcVnImage;	(* Source image *)
		ipDestImage	:	REFERENCE TO ITcVnImage;	(* Destination image (An appropriate image will be created if required.) *)
		fAngleDeg	:	LREAL;	(* Rotation angle in degree (positive: counter-clockwise, negative: clockwise) *)
		bAdjustDestSize	:	BOOL;	(* If true, ipDestImage size is adjusted so that the whole rotated ipSrcImage is contained. Otherwise, ipDestImage size is set to ipSrcImage size. *)
		hrPrev	:	HRESULT;	(* HRESULT indicating the result of previous operations (If SUCCEEDED(hrPrev) equals false, no operation is executed.) *)
	END_VAR

END_FUNCTION

// Functions/Geometric and Coordinate Transformations/F_VN_RotateImageExp2

	{attribute 'TcIecLibraryType'}
	{attribute 'external_name' := 'F_VN_RotateImageExp2_GUID_7D0B9B63_6D0D_0B6C_6539_4698A9F08E11'}
	(* Rotate an image by an individual rotation angle in degrees. (expert function) *)
	FUNCTION F_VN_RotateImageExp2 : HRESULT
	VAR_INPUT
		ipSrcImage	:	ITcVnImage;	(* Source image *)
		ipDestImage	:	REFERENCE TO ITcVnImage;	(* Destination image (An appropriate image will be created if required.) *)
		fAngleDeg	:	LREAL;	(* Rotation angle in degree (positive: counter-clockwise, negative: clockwise) *)
		bAdjustDestSize	:	BOOL;	(* If true, ipDestImage size is adjusted so that the whole rotated ipSrcImage is contained. Otherwise, ipDestImage size is set to ipSrcImage size. *)
		eInterpolationType	:	ETcVnInterpolationType;	(* Interpolation method *)
		eBorderInterpolation	:	ETcVnBorderInterpolationMethod;	(* Border interpolation method (ISOLATED not supported) *)
		aBorderValue	:	REFERENCE TO TcVnVector4_LREAL;	(* Border value, if CONSTANT is used *)
		hrPrev	:	HRESULT;	(* HRESULT indicating the result of previous operations (If SUCCEEDED(hrPrev) equals false, no operation is executed.) *)
	END_VAR

END_FUNCTION

// Functions/Geometric and Coordinate Transformations/F_VN_WarpAffineExp

	{attribute 'TcIecLibraryType'}
	{attribute 'external_name' := 'F_VN_WarpAffineExp_GUID_1D3796C5_DE37_0D70_4E15_B2E56F13E25E'}
	(* Apply an affine transformation to an image. (expert function) *)
	FUNCTION F_VN_WarpAffineExp : HRESULT
	VAR_INPUT
		ipSrcImage	:	ITcVnImage;	(* Source image *)
		ipDestImage	:	REFERENCE TO ITcVnImage;	(* Destination image (An appropriate image will be created if required.) *)
		aTransformationMatrix	:	REFERENCE TO TcVnMatrix2x3_LREAL;	(* Affine transformation matrix *)
		nDestWidth	:	UDINT;	(* Width of the destination image *)
		nDestHeight	:	UDINT;	(* Height of the destination image *)
		eInterpolationType	:	ETcVnInterpolationType;	(* Interpolation method *)
		bWarpInverse	:	BOOL;	(* Handle aTransformationMatrix as the inverse transformation *)
		eBorderInterpolation	:	ETcVnBorderInterpolationMethod;	(* Border interpolation method (ISOLATED not supported) *)
		fBorderValue	:	LREAL;	(* Border value, if CONSTANT is used *)
		hrPrev	:	HRESULT;	(* HRESULT indicating the result of previous operations (If SUCCEEDED(hrPrev) equals false, no operation is executed.) *)
	END_VAR

END_FUNCTION

// Functions/Geometric and Coordinate Transformations/F_VN_WarpAffine_Container

	{attribute 'TcIecLibraryType'}
	{attribute 'external_name' := 'F_VN_WarpAffine_Container_GUID_455E81FB_A540_0FCD_7BE9_3DE9B2BA6451'}
	(* Apply an affine transformation to a container of 2D points. *)
	FUNCTION F_VN_WarpAffine_Container : HRESULT
	VAR_INPUT
		ipSrcPoints	:	ITcVnContainer;	(* Source points (ContainerType_Vector_TcVnPoint2_DINT or ContainerType_Vector_TcVnPoint2_REAL or ContainerType_Vector_TcVnPoint2_LREAL) *)
		ipDestPoints	:	REFERENCE TO ITcVnContainer;	(* Returns the transformed points (same type ID as ipSrcPoints; Non-zero interface pointers are reused.) *)
		aTransformationMatrix	:	REFERENCE TO TcVnMatrix2x3_LREAL;	(* Affine transformation matrix *)
		hrPrev	:	HRESULT;	(* HRESULT indicating the result of previous operations (If SUCCEEDED(hrPrev) equals false, no operation is executed.) *)
	END_VAR

END_FUNCTION

// Functions/Geometric and Coordinate Transformations/F_VN_WarpAffine_Point

	{attribute 'TcIecLibraryType'}
	{attribute 'external_name' := 'F_VN_WarpAffine_Point_GUID_F499FEDB_995B_0AB5_479C_FCE235D0B403'}
	(* Apply an affine transformation to a 2D point. *)
	FUNCTION F_VN_WarpAffine_Point : HRESULT
	VAR_INPUT
		aSrcPoint	:	REFERENCE TO TcVnPoint2_LREAL;	(* Source point *)
		aDestPoint	:	REFERENCE TO TcVnPoint2_LREAL;	(* Destination point *)
		aTransformationMatrix	:	REFERENCE TO TcVnMatrix2x3_LREAL;	(* Affine transformation matrix *)
		hrPrev	:	HRESULT;	(* HRESULT indicating the result of previous operations (If SUCCEEDED(hrPrev) equals false, no operation is executed.) *)
	END_VAR

END_FUNCTION

// Functions/Geometric and Coordinate Transformations/F_VN_WarpAffine_Rectangle

	{attribute 'TcIecLibraryType'}
	{attribute 'external_name' := 'F_VN_WarpAffine_Rectangle_GUID_A4F17C87_D410_09C6_4083_D1094D7549FA'}
	(* Use an affine transform to warp a rectangle. *)
	FUNCTION F_VN_WarpAffine_Rectangle : HRESULT
	VAR_INPUT
		nTopLeftX	:	UDINT;	(* x coordinate of the top left corner *)
		nTopLeftY	:	UDINT;	(* y coordinate of the top left corner *)
		nBottomRightX	:	UDINT;	(* x coordinate of the bottom right corner *)
		nBottomRightY	:	UDINT;	(* y coordinate of the bottom right corner *)
		ipDestPoints	:	REFERENCE TO ITcVnContainer;	(* Returns the 4 transformed points (ContainerType_Vector_TcVnPoint2_REAL) *)
		aTransformationMatrix	:	REFERENCE TO TcVnMatrix2x3_LREAL;	(* Affine transformation matrix *)
		hrPrev	:	HRESULT;	(* HRESULT indicating the result of previous operations (If SUCCEEDED(hrPrev) equals false, no operation is executed.) *)
	END_VAR

END_FUNCTION

// Functions/Geometric and Coordinate Transformations/F_VN_WarpPerspective

	{attribute 'TcIecLibraryType'}
	{attribute 'external_name' := 'F_VN_WarpPerspective_GUID_02ABC27A_AE98_0CBA_57E7_0B0493B09EA2'}
	(* Apply a perspective transformation to an image. *)
	FUNCTION F_VN_WarpPerspective : HRESULT
	VAR_INPUT
		ipSrcImage	:	ITcVnImage;	(* Source image *)
		ipDestImage	:	REFERENCE TO ITcVnImage;	(* Destination image (An appropriate image will be created if required.) *)
		aTransformationMatrix	:	REFERENCE TO TcVnMatrix3x3_LREAL;	(* Perspective transformation matrix *)
		hrPrev	:	HRESULT;	(* HRESULT indicating the result of previous operations (If SUCCEEDED(hrPrev) equals false, no operation is executed.) *)
	END_VAR

END_FUNCTION

// Functions/Geometric and Coordinate Transformations/F_VN_WarpPerspective_Container

	{attribute 'TcIecLibraryType'}
	{attribute 'external_name' := 'F_VN_WarpPerspective_Container_GUID_097EA9FE_890E_034A_71DB_5AD3771EB640'}
	(* Apply a perspective transformation to a container of 2D points. *)
	FUNCTION F_VN_WarpPerspective_Container : HRESULT
	VAR_INPUT
		ipSrcPoints	:	ITcVnContainer;	(* Source points (ContainerType_Vector_TcVnPoint2_DINT or ContainerType_Vector_TcVnPoint2_REAL or ContainerType_Vector_TcVnPoint2_LREAL) *)
		ipDestPoints	:	REFERENCE TO ITcVnContainer;	(* Returns the transformed points (same type ID as ipSrcPoints; Non-zero interface pointers are reused.) *)
		aTransformationMatrix	:	REFERENCE TO TcVnMatrix3x3_LREAL;	(* Perspective transformation matrix *)
		hrPrev	:	HRESULT;	(* HRESULT indicating the result of previous operations (If SUCCEEDED(hrPrev) equals false, no operation is executed.) *)
	END_VAR

END_FUNCTION

// Functions/Geometric and Coordinate Transformations/F_VN_WarpPerspectiveExp

	{attribute 'TcIecLibraryType'}
	{attribute 'external_name' := 'F_VN_WarpPerspectiveExp_GUID_F9FDE0D0_7EBE_09AF_42AE_C4EBF9FF834C'}
	(* Apply a perspective transformation to an image. (expert function) *)
	FUNCTION F_VN_WarpPerspectiveExp : HRESULT
	VAR_INPUT
		ipSrcImage	:	ITcVnImage;	(* Source image *)
		ipDestImage	:	REFERENCE TO ITcVnImage;	(* Destination image (An appropriate image will be created if required.) *)
		aTransformationMatrix	:	REFERENCE TO TcVnMatrix3x3_LREAL;	(* Perspective transformation matrix *)
		nDestWidth	:	UDINT;	(* Width of the destination image *)
		nDestHeight	:	UDINT;	(* Height of the destination image *)
		eInterpolationType	:	ETcVnInterpolationType;	(* Interpolation method *)
		bWarpInverse	:	BOOL;	(* Handle aTransformationMatrix as the inverse transformation *)
		eBorderInterpolation	:	ETcVnBorderInterpolationMethod;	(* Border interpolation method (ISOLATED not supported) *)
		fBorderValue	:	LREAL;	(* Border value, if CONSTANT is used *)
		hrPrev	:	HRESULT;	(* HRESULT indicating the result of previous operations (If SUCCEEDED(hrPrev) equals false, no operation is executed.) *)
	END_VAR

END_FUNCTION

// Functions/Geometric and Coordinate Transformations/F_VN_WarpPerspective_Point

	{attribute 'TcIecLibraryType'}
	{attribute 'external_name' := 'F_VN_WarpPerspective_Point_GUID_F223DF96_56E3_0B0C_5D9D_3E66FB302F8A'}
	(* Apply a perspective transformation to a 2D point. *)
	FUNCTION F_VN_WarpPerspective_Point : HRESULT
	VAR_INPUT
		aSrcPoint	:	REFERENCE TO TcVnPoint2_LREAL;	(* Source point *)
		aDestPoint	:	REFERENCE TO TcVnPoint2_LREAL;	(* Destination point *)
		aTransformationMatrix	:	REFERENCE TO TcVnMatrix3x3_LREAL;	(* Perspective transformation matrix *)
		hrPrev	:	HRESULT;	(* HRESULT indicating the result of previous operations (If SUCCEEDED(hrPrev) equals false, no operation is executed.) *)
	END_VAR

END_FUNCTION

// Functions/Geometric and Coordinate Transformations/F_VN_WarpPerspective_Rectangle

	{attribute 'TcIecLibraryType'}
	{attribute 'external_name' := 'F_VN_WarpPerspective_Rectangle_GUID_044EE11D_B6DB_0F36_463E_73E455BB4E23'}
	(* Use a perspective transform to warp a rectangle. *)
	FUNCTION F_VN_WarpPerspective_Rectangle : HRESULT
	VAR_INPUT
		nTopLeftX	:	UDINT;	(* x coordinate of the top left corner *)
		nTopLeftY	:	UDINT;	(* y coordinate of the top left corner *)
		nBottomRightX	:	UDINT;	(* x coordinate of the bottom right corner *)
		nBottomRightY	:	UDINT;	(* y coordinate of the bottom right corner *)
		ipDestPoints	:	REFERENCE TO ITcVnContainer;	(* Returns the 4 transformed points (ContainerType_Vector_TcVnPoint2_REAL) *)
		aTransformationMatrix	:	REFERENCE TO TcVnMatrix3x3_LREAL;	(* Perspective transformation matrix *)
		hrPrev	:	HRESULT;	(* HRESULT indicating the result of previous operations (If SUCCEEDED(hrPrev) equals false, no operation is executed.) *)
	END_VAR

END_FUNCTION

// Functions/Image Color and Contrast Processing/F_VN_ApplyColorMap

	{attribute 'TcIecLibraryType'}
	{attribute 'external_name' := 'F_VN_ApplyColorMap_GUID_928F246E_5D28_0E29_5FCC_94F262C9C14B'}
	(* Apply a color map to a gray-level image. *)
	FUNCTION F_VN_ApplyColorMap : HRESULT
	VAR_INPUT
		ipSrcImage	:	ITcVnImage;	(* Source image (TCVN_ET_USINT or TCVN_ET_UINT, 1 channel) *)
		ipDestImage	:	REFERENCE TO ITcVnImage;	(* Returns the colored image (TCVN_ET_USINT, 3 channel. An appropriate image will be created if required.) *)
		ipColorMap	:	ITcVnContainer;	(* Color map to be applied to ipSrcImage (ContainerType_Vector_TcVnVector3_REAL with 256 or 65536 elements, dependent on ipSrcImage type). Can be either custom or created with F_VN_GenerateColorMap. *)
		hrPrev	:	HRESULT;	(* HRESULT indicating the result of previous operations (If SUCCEEDED(hrPrev) equals false, no operation is executed.) *)
	END_VAR

END_FUNCTION

// Functions/Image Color and Contrast Processing/F_VN_GenerateColorMap

	{attribute 'TcIecLibraryType'}
	{attribute 'external_name' := 'F_VN_GenerateColorMap_GUID_8C5C9B2E_64E8_0746_749F_E4647C39DBCC'}
	(* Generates a pre-defined color map. *)
	FUNCTION F_VN_GenerateColorMap : HRESULT
	VAR_INPUT
		ipColorMap	:	REFERENCE TO ITcVnContainer;	(* Returns the color map (ContainerType_Vector_TcVnVector3_REAL with 256 or 65536 elements) *)
		eColorMap	:	ETcVnColorMap;	(* Selects a color map (similar to GNU Octave/MATLAB types) *)
		eColorMapSize	:	ETcVnColorMapSize;	(* Defines how many elements the generated color map should have *)
		hrPrev	:	HRESULT;	(* HRESULT indicating the result of previous operations (If SUCCEEDED(hrPrev) equals false, no operation is executed.) *)
	END_VAR

END_FUNCTION

// Functions/Image Color and Contrast Processing/F_VN_ApplyLut

	{attribute 'TcIecLibraryType'}
	{attribute 'external_name' := 'F_VN_ApplyLut_GUID_903DA918_CE30_0A02_501C_F9B2F836B055'}
	(* Apply a lookup table to an image to manipulate its colors. *)
	FUNCTION F_VN_ApplyLut : HRESULT
	VAR_INPUT
		ipSrcImage	:	ITcVnImage;	(* Source image (1-4 channels of 8 or 16 bit types SINT, USINT, INT, UINT) *)
		ipDestImage	:	REFERENCE TO ITcVnImage;	(* Returns the result image (same size, type and channels as ipSrcImage. An appropriate image will be created if required.) *)
		ipLut	:	ITcVnContainer;	(* Lookup table with elements matching ipSrcImage type and either 256 (8 bit images) or 65536 (16 bit images) elements. E.g. ContainerType_Vector_USINT for 1-4 channel USINT image (in this case, the same lookup values are used for each channel) or ContainerType_Vector_TcVnVector3_USINT for a 3 channel USINT image (in this case, each channel uses an individual lookup value).
						 *)
		hrPrev	:	HRESULT;	(* HRESULT indicating the result of previous operations (If SUCCEEDED(hrPrev) equals false, no operation is executed.) *)
	END_VAR

END_FUNCTION

// Functions/Image Color and Contrast Processing/F_VN_Clahe

	{attribute 'TcIecLibraryType'}
	{attribute 'external_name' := 'F_VN_Clahe_GUID_A2DC4928_144D_03A4_6714_ECC6B4ABE99B'}
	(* Apply Constrast Limited Adaptive Histogram Equalization. This applies local histogram equalization to individual tiles. *)
	FUNCTION F_VN_Clahe : HRESULT
	VAR_INPUT
		ipSrcImage	:	ITcVnImage;	(* Source image (TCVN_ET_USINT or TCVN_ET_UINT, 1 channel) *)
		ipDestImage	:	REFERENCE TO ITcVnImage;	(* Returns the resulting image (An appropriate image will be created if required.) *)
		hrPrev	:	HRESULT;	(* HRESULT indicating the result of previous operations (If SUCCEEDED(hrPrev) equals false, no operation is executed.) *)
	END_VAR

END_FUNCTION

// Functions/Image Color and Contrast Processing/F_VN_ClaheExp

	{attribute 'TcIecLibraryType'}
	{attribute 'external_name' := 'F_VN_ClaheExp_GUID_18E07C8A_7F67_03C2_5B68_ACE15477BAB5'}
	(* Apply Constrast Limited Adaptive Histogram Equalization. This applies local histogram equalization to individual tiles. (expert function) *)
	FUNCTION F_VN_ClaheExp : HRESULT
	VAR_INPUT
		ipSrcImage	:	ITcVnImage;	(* Source image (TCVN_ET_USINT or TCVN_ET_UINT, 1 channel) *)
		ipDestImage	:	REFERENCE TO ITcVnImage;	(* Returns the resulting image (An appropriate image will be created if required.) *)
		fClipLimit	:	LREAL;	(* Threshold for contrast limit (set to <= 0 to disable clipping) *)
		nTilesX	:	UDINT;	(* Number of tiles in x direction *)
		nTilesY	:	UDINT;	(* Number of tiles in y direction *)
		hrPrev	:	HRESULT;	(* HRESULT indicating the result of previous operations (If SUCCEEDED(hrPrev) equals false, no operation is executed.) *)
	END_VAR

END_FUNCTION

// Functions/Image Color and Contrast Processing/F_VN_ConvertColorSpace

	{attribute 'TcIecLibraryType'}
	{attribute 'external_name' := 'F_VN_ConvertColorSpace_GUID_F4663C0B_5492_0ADD_5399_51D6D0FA574F'}
	(* Convert image from one color space to another. *)
	FUNCTION F_VN_ConvertColorSpace : HRESULT
	VAR_INPUT
		ipSrcImage	:	ITcVnImage;	(* Source image *)
		ipDestImage	:	REFERENCE TO ITcVnImage;	(* Destination image (An appropriate destination image will be created if required.) *)
		eTransform	:	ETcVnColorSpaceTransform;	(* Transforms to be applied *)
		hrPrev	:	HRESULT;	(* HRESULT indicating the result of previous operations (If SUCCEEDED(hrPrev) equals false, no operation is executed.) *)
	END_VAR

END_FUNCTION

// Functions/Image Color and Contrast Processing/F_VN_GenerateCustomColorMap

	{attribute 'TcIecLibraryType'}
	{attribute 'external_name' := 'F_VN_GenerateCustomColorMap_GUID_E8688580_DF85_076C_6503_2DD9DD62FECB'}
	(* Generate a custom color map by interpolating between user defined colors (equally distributed, linear for each channel). *)
	FUNCTION F_VN_GenerateCustomColorMap : HRESULT
	VAR_INPUT
		ipColorMap	:	REFERENCE TO ITcVnContainer;	(* Returns the color map (ContainerType_Vector_TcVnVector3_REAL with 256 or 65536 elements) *)
		ipInitialColors	:	ITcVnContainer;	(* User defined colors (ContainerType_Vector_TcVnVector3_REAL, at least 2 elements) *)
		eColorMapSize	:	ETcVnColorMapSize;	(* Defines how many elements the generated color map should have *)
		hrPrev	:	HRESULT;	(* HRESULT indicating the result of previous operations (If SUCCEEDED(hrPrev) equals false, no operation is executed.) *)
	END_VAR

END_FUNCTION

// Functions/Image Color and Contrast Processing/F_VN_Histogram

	{attribute 'TcIecLibraryType'}
	{attribute 'external_name' := 'F_VN_Histogram_GUID_84297A6C_7A54_07A2_45AB_3D98EC25B86B'}
	(* Calculate the (multi-channel) histogram of an image. *)
	FUNCTION F_VN_Histogram : HRESULT
	VAR_INPUT
		ipSrcImage	:	ITcVnImage;	(* Source image *)
		ipDestHistogram	:	REFERENCE TO ITcVnContainer;	(* Returns a container with a multi-channel histogram, where every channel is represented as a vector of UDINT (ContainerType_Vector_Vector_UDINT. Non-zero interface pointers are reused.) *)
		hrPrev	:	HRESULT;	(* HRESULT indicating the result of previous operations (If SUCCEEDED(hrPrev) equals false, no operation is executed.) *)
	END_VAR

END_FUNCTION

// Functions/Image Color and Contrast Processing/F_VN_HistogramExp

	{attribute 'TcIecLibraryType'}
	{attribute 'external_name' := 'F_VN_HistogramExp_GUID_0F031BD5_943B_00D5_637C_50BDFC802233'}
	(* Calculate the (multi-channel) histogram of an image. (expert function) *)
	FUNCTION F_VN_HistogramExp : HRESULT
	VAR_INPUT
		ipSrcImage	:	ITcVnImage;	(* Source image *)
		ipDestHistogram	:	REFERENCE TO ITcVnContainer;	(* Returns a container with a multi-channel histogram, where every channel is represented as a vector of UDINT (ContainerType_Vector_Vector_UDINT. Non-zero interface pointers are reused.) *)
		nBins	:	REFERENCE TO UDINT;	(* Desired number of bins or 0 to keep the default for the corresponding image format (in) and default number of bins (out) *)
		fLowerBound	:	REFERENCE TO LREAL;	(* Lower (inclusive) boundary of the 0-th histogram bin (in), or receive the default if fLowerBound AND fUpperBound are set to 0 (out) *)
		fUpperBound	:	REFERENCE TO LREAL;	(* Upper (exclusive) boundary of the last histogram bin nBins-1 (in), or receive the default if fLowerBound AND fUpperBound are set to 0 (out) *)
		ipMask	:	ITcVnImage;	(* Source image mask (TCVN_ET_USINT, 1 channel. Mask is optional, set to 0 if not required.) *)
		hrPrev	:	HRESULT;	(* HRESULT indicating the result of previous operations (If SUCCEEDED(hrPrev) equals false, no operation is executed.) *)
	END_VAR

END_FUNCTION

// Functions/Image Color and Contrast Processing/F_VN_HistogramEqualization

